(* Logix 5000 project; controller ACMI_PLC vendor 1 type 14 code 101 rev 19.11; software revision 19.01; part 17 of 18 *)
(* tags used below, declared in another part *)
   A : DINT;
   ACMI_BR_CNT : DINT;
   ACMI_Stat_Size : INT;
   ACMI_TO_CNT : DINT;
   ADCA : DINT;
   ADCB : DINT;
   B : DINT;
   Beam_MaxQ : DINT;
   Beam_MinQ : DINT;
   Beam_Q : DINT;
   BR_Stack : DINT[7200];
   BR_Stack_MAX : DINT;
   BR_Stack_Sum : DINT;
   BR_Stack_Top : DINT;
   BSSS_CLOSED : ALIAS FOR PointIONet:7:I.Pt00Data;
   BYPASS_KEY : ALIAS FOR PointIONet:5:I.Pt07Data;
   FAULT_BEAM_BL : BOOL;
   FAULT_BEAM_HI : BOOL;
   FAULT_BEAM_LO : BOOL;
   FAULT_BR_ACC : BOOL;
   FAULT_CODE : DINT;
   FAULT_QOW1 : BOOL;
   FAULT_ST1_AB_HI : BOOL;
   FAULT_ST1_AB_LO : BOOL;
   FAULT_ST1_BA_HI : BOOL;
   FAULT_ST1_BA_LO : BOOL;
   FAULT_ST1_BLA : BOOL;
   FAULT_ST1_BLB : BOOL;
   FAULT_ST1_QAT : BOOL;
   FAULT_ST2_AB_HI : BOOL;
   FAULT_ST2_AB_LO : BOOL;
   FAULT_ST2_BA_HI : BOOL;
   FAULT_ST2_BA_LO : BOOL;
   FAULT_ST2_BLA : BOOL;
   FAULT_ST2_BLB : BOOL;
   FAULT_ST2_QAT : BOOL;
   FAULT_TO_ACC : BOOL;
   FAULT_TWB : BOOL;
   FAULT_WDT : BOOL;
   Initialize : BOOL;
   LBSS_CLOSED : ALIAS FOR PointIONet:7:I.Pt01Data;
   ST1_MaxQ : DINT;
   ST1_MinQ : DINT;
   ST1_QAB : DINT;
   ST1_QBA : DINT;
   ST2_MaxQ : DINT;
   ST2_MinQ : DINT;
   ST2_QAB : DINT;
   ST2_QBA : DINT;
   ST_HI_FAULT : BOOL;
   ST_LO_FAULT : BOOL;
   ST_Size : BOOL;
   ST_Type : BOOL;
   Stack_Size : DINT;
   TO_Cntr : COUNTER;
   TO_DISABLED : ALIAS FOR PointIONet:7:I.Pt03Data;
   TO_Stack : DINT[120];
   TO_Stack_MAX : DINT;
   TO_Stack_Size : DINT;
   TO_Stack_Sum : DINT;
   TO_Stack_Top : DINT;
   TO_Status_Error : BOOL;
   Update_ST1_QAB : BOOL;
   Update_ST1_QBA : BOOL;
   Update_ST2_QAB : BOOL;
   Update_ST2_QBA : BOOL;
   Zero : DINT[7200];

        [22].Hist[3812] := 1, [22].Hist[3815] := 1, [22].Hist[3816] := 1, [22].Hist[3817] := 1, [22].Hist[3819] := 1, [22].Hist[3820] := 1, [22].Hist[3824] := 1, [22].Hist[3825] := 1, [22].Hist[3828] := 1, [22].Hist[3832] := 1, [22].Hist[3835] := 1, [22].Hist[3836] := 1, [22].Hist[3839] := 1, [22].Hist[3840] := 1, [22].Hist[3844] := 1, [22].Hist[3848] := 1, [22].Hist[3852] := 1, [22].Hist[3853] := 1, [22].Hist[3855] := 1, [22].Hist[3856] := 1, [22].Hist[3859] := 1, [22].Hist[3860] := 1, [22].Hist[3864] := 1, [22].Hist[3868] := 1, [22].Hist[3869] := 1, [22].Hist[3872] := 1, [22].Hist[3875] := 1, [22].Hist[3876] := 1, [22].Hist[3880] := 1, [22].Hist[3881] := 1, [22].Hist[3883] := 1, [22].Hist[3884] := 1, [22].Hist[3885] := 1, [22].Hist[3888] := 1, [22].Hist[3891] := 1, [22].Hist[3892] := 1, [22].Hist[3896] := 1, [22].Hist[3900] := 1, [22].Hist[3901] := 1, [22].Hist[3903] := 1, [22].Hist[3904] := 1, [22].Hist[3908] := 1, [22].Hist[3912] := 1, [22].Hist[3916] := 1, [22].Hist[3917] := 1, [22].Hist[3920] := 1, [22].Hist[3921] := 1, [22].Hist[3924] := 1, [22].Hist[3927] := 1, [22].Hist[3928] := 1, [22].Hist[3929] := 1, [22].Hist[3932] := 1, [22].Hist[3935] := 1, [22].Hist[3936] := 1, [22].Hist[3940] := 1, [22].Hist[3944] := 1, [22].Hist[3948] := 1, [22].Hist[3952] := 1, [22].Hist[3953] := 1, [22].Hist[3955] := 1,
        [22].Hist[3956] := 1, [22].Hist[3960] := 1, [22].Hist[3964] := 1, [22].Hist[3967] := 1, [22].Hist[3968] := 1, [22].Hist[3969] := 1, [22].Hist[3972] := 1, [22].Hist[3976] := 1, [22].Hist[3977] := 1, [22].Hist[3980] := 1, [22].Hist[3984] := 1, [22].Hist[3988] := 1, [22].Hist[3992] := 1, [22].Hist[3995] := 1, [22].Hist[3996] := 1, [22].Hist[4000] := 1, [22].Hist[4004] := 1, [22].Hist[4008] := 1, [22].Hist[4012] := 1, [22].Hist[4013] := 1, [22].Hist[4016] := 1, [22].Hist[4020] := 1, [22].Hist[4024] := 1, [22].Hist[4025] := 1, [22].Hist[4028] := 1, [22].Hist[4029] := 1, [22].Hist[4032] := 1, [22].Hist[4036] := 1, [22].Hist[4040] := 1, [22].Hist[4044] := 1, [22].Hist[4047] := 1, [22].Hist[4048] := 1, [22].Hist[4052] := 1, [22].Hist[4056] := 1, [22].Hist[4057] := 1, [22].Hist[4060] := 1, [22].Hist[4061] := 1, [22].Hist[4063] := 1, [22].Hist[4064] := 1, [22].Hist[4068] := 1, [22].Hist[4072] := 1, [22].Hist[4076] := 1, [22].Hist[4080] := 1, [22].Hist[4081] := 1, [22].Hist[4084] := 1, [22].Hist[4087] := 1, [22].Hist[4088] := 1, [22].Hist[4092] := 1, [22].Top := 3827, [22].Sum := 1635, [23].Hist[3] := 1, [23].Hist[5] := 1, [23].Hist[9] := 1, [23].Hist[17] := 1, [23].Hist[19] := 1, [23].Hist[29] := 1, [23].Hist[31] := 1, [23].Hist[37] := 1, [23].Hist[39] := 1, [23].Hist[41] := 1,
        [23].Hist[51] := 1, [23].Hist[55] := 1, [23].Hist[63] := 1, [23].Hist[67] := 1, [23].Hist[73] := 1, [23].Hist[77] := 1, [23].Hist[81] := 1, [23].Hist[89] := 1, [23].Hist[95] := 1, [23].Hist[107] := 1, [23].Hist[115] := 1, [23].Hist[117] := 1, [23].Hist[125] := 1, [23].Hist[127] := 1, [23].Hist[135] := 1, [23].Hist[153] := 1, [23].Hist[155] := 1, [23].Hist[165] := 1, [23].Hist[179] := 1, [23].Hist[187] := 1, [23].Hist[199] := 1, [23].Hist[213] := 1, [23].Hist[223] := 1, [23].Hist[239] := 1, [23].Hist[243] := 1, [23].Hist[251] := 1, [23].Hist[253] := 1, [23].Hist[255] := 1, [23].Hist[257] := 1, [23].Hist[261] := 1, [23].Hist[271] := 1, [23].Hist[277] := 1, [23].Hist[291] := 1, [23].Hist[293] := 1, [23].Hist[301] := 1, [23].Hist[307] := 1, [23].Hist[313] := 1, [23].Hist[317] := 1, [23].Hist[321] := 1, [23].Hist[323] := 1, [23].Hist[331] := 1, [23].Hist[337] := 1, [23].Hist[341] := 1, [23].Hist[347] := 1, [23].Hist[351] := 1, [23].Hist[353] := 1, [23].Hist[359] := 1, [23].Hist[361] := 1, [23].Hist[365] := 1, [23].Hist[367] := 1, [23].Hist[369] := 1, [23].Hist[373] := 1, [23].Hist[405] := 1, [23].Hist[413] := 1, [23].Hist[417] := 1, [23].Hist[423] := 1, [23].Hist[425] := 1, [23].Hist[429] := 1, [23].Hist[433] := 1, [23].Hist[441] := 1,
        [23].Hist[443] := 1, [23].Hist[445] := 1, [23].Hist[447] := 1, [23].Hist[459] := 1, [23].Hist[471] := 1, [23].Hist[473] := 1, [23].Hist[491] := 1, [23].Hist[501] := 1, [23].Hist[509] := 1, [23].Hist[515] := 1, [23].Hist[519] := 1, [23].Hist[527] := 1, [23].Hist[529] := 1, [23].Hist[537] := 1, [23].Hist[543] := 1, [23].Hist[547] := 1, [23].Hist[553] := 1, [23].Hist[557] := 1, [23].Hist[559] := 1, [23].Hist[567] := 1, [23].Hist[569] := 1, [23].Hist[581] := 1, [23].Hist[601] := 1, [23].Hist[611] := 1, [23].Hist[613] := 1, [23].Hist[619] := 1, [23].Hist[621] := 1, [23].Hist[629] := 1, [23].Hist[637] := 1, [23].Hist[647] := 1, [23].Hist[663] := 1, [23].Hist[669] := 1, [23].Hist[677] := 1, [23].Hist[679] := 1, [23].Hist[689] := 1, [23].Hist[691] := 1, [23].Hist[693] := 1, [23].Hist[695] := 1, [23].Hist[709] := 1, [23].Hist[723] := 1, [23].Hist[737] := 1, [23].Hist[741] := 1, [23].Hist[747] := 1, [23].Hist[749] := 1, [23].Hist[751] := 1, [23].Hist[761] := 1, [23].Hist[767] := 1, [23].Hist[773] := 1, [23].Hist[777] := 1, [23].Hist[799] := 1, [23].Hist[801] := 1, [23].Hist[825] := 1, [23].Hist[827] := 1, [23].Hist[829] := 1, [23].Hist[841] := 1, [23].Hist[847] := 1, [23].Hist[853] := 1, [23].Hist[859] := 1, [23].Hist[863] := 1, [23].Hist[865] := 1,
        [23].Hist[867] := 1, [23].Hist[875] := 1, [23].Hist[877] := 1, [23].Hist[879] := 1, [23].Hist[881] := 1, [23].Hist[883] := 1, [23].Hist[891] := 1, [23].Hist[893] := 1, [23].Hist[911] := 1, [23].Hist[923] := 1, [23].Hist[927] := 1, [23].Hist[935] := 1, [23].Hist[943] := 1, [23].Hist[945] := 1, [23].Hist[947] := 1, [23].Hist[961] := 1, [23].Hist[969] := 1, [23].Hist[973] := 1, [23].Hist[983] := 1, [23].Hist[985] := 1, [23].Hist[987] := 1, [23].Hist[995] := 1, [23].Hist[1015] := 1, [23].Hist[1021] := 1, [23].Hist[1041] := 1, [23].Hist[1045] := 1, [23].Hist[1047] := 1, [23].Hist[1049] := 1, [23].Hist[1053] := 1, [23].Hist[1057] := 1, [23].Hist[1059] := 1, [23].Hist[1061] := 1, [23].Hist[1065] := 1, [23].Hist[1073] := 1, [23].Hist[1077] := 1, [23].Hist[1079] := 1, [23].Hist[1085] := 1, [23].Hist[1093] := 1, [23].Hist[1095] := 1, [23].Hist[1101] := 1, [23].Hist[1109] := 1, [23].Hist[1125] := 1, [23].Hist[1129] := 1, [23].Hist[1135] := 1, [23].Hist[1137] := 1, [23].Hist[1141] := 1, [23].Hist[1145] := 1, [23].Hist[1149] := 1, [23].Hist[1155] := 1, [23].Hist[1167] := 1, [23].Hist[1175] := 1, [23].Hist[1181] := 1, [23].Hist[1185] := 1, [23].Hist[1195] := 1, [23].Hist[1209] := 1, [23].Hist[1217] := 1, [23].Hist[1235] := 1, [23].Hist[1237] := 1, [23].Hist[1239] := 1, [23].Hist[1245] := 1,
        [23].Hist[1257] := 1, [23].Hist[1265] := 1, [23].Hist[1269] := 1, [23].Hist[1271] := 1, [23].Hist[1277] := 1, [23].Hist[1279] := 1, [23].Hist[1281] := 1, [23].Hist[1291] := 1, [23].Hist[1299] := 1, [23].Hist[1307] := 1, [23].Hist[1325] := 1, [23].Hist[1329] := 1, [23].Hist[1335] := 1, [23].Hist[1347] := 1, [23].Hist[1349] := 1, [23].Hist[1351] := 1, [23].Hist[1357] := 1, [23].Hist[1361] := 1, [23].Hist[1365] := 1, [23].Hist[1383] := 1, [23].Hist[1389] := 1, [23].Hist[1397] := 1, [23].Hist[1401] := 1, [23].Hist[1407] := 1, [23].Hist[1411] := 1, [23].Hist[1413] := 1, [23].Hist[1419] := 1, [23].Hist[1429] := 1, [23].Hist[1437] := 1, [23].Hist[1451] := 1, [23].Hist[1469] := 1, [23].Hist[1471] := 1, [23].Hist[1477] := 1, [23].Hist[1483] := 1, [23].Hist[1487] := 1, [23].Hist[1489] := 1, [23].Hist[1491] := 1, [23].Hist[1495] := 1, [23].Hist[1497] := 1, [23].Hist[1501] := 1, [23].Hist[1511] := 1, [23].Hist[1515] := 1, [23].Hist[1517] := 1, [23].Hist[1519] := 1, [23].Hist[1521] := 1, [23].Hist[1535] := 1, [23].Hist[1539] := 1, [23].Hist[1545] := 1, [23].Hist[1547] := 1, [23].Hist[1551] := 1, [23].Hist[1555] := 1, [23].Hist[1557] := 1, [23].Hist[1559] := 1, [23].Hist[1563] := 1, [23].Hist[1565] := 1, [23].Hist[1569] := 1, [23].Hist[1581] := 1, [23].Hist[1593] := 1, [23].Hist[1605] := 1, [23].Hist[1611] := 1,
        [23].Hist[1617] := 1, [23].Hist[1627] := 1, [23].Hist[1651] := 1, [23].Hist[1653] := 1, [23].Hist[1655] := 1, [23].Hist[1669] := 1, [23].Hist[1677] := 1, [23].Hist[1679] := 1, [23].Hist[1681] := 1, [23].Hist[1683] := 1, [23].Hist[1685] := 1, [23].Hist[1691] := 1, [23].Hist[1697] := 1, [23].Hist[1709] := 1, [23].Hist[1715] := 1, [23].Hist[1717] := 1, [23].Hist[1721] := 1, [23].Hist[1731] := 1, [23].Hist[1737] := 1, [23].Hist[1741] := 1, [23].Hist[1747] := 1, [23].Hist[1753] := 1, [23].Hist[1769] := 1, [23].Hist[1771] := 1, [23].Hist[1779] := 1, [23].Hist[1783] := 1, [23].Hist[1785] := 1, [23].Hist[1793] := 1, [23].Hist[1805] := 1, [23].Hist[1807] := 1, [23].Hist[1811] := 1, [23].Hist[1819] := 1, [23].Hist[1821] := 1, [23].Hist[1825] := 1, [23].Hist[1827] := 1, [23].Hist[1833] := 1, [23].Hist[1839] := 1, [23].Hist[1843] := 1, [23].Hist[1849] := 1, [23].Hist[1851] := 1, [23].Hist[1857] := 1, [23].Hist[1863] := 1, [23].Hist[1877] := 1, [23].Hist[1879] := 1, [23].Hist[1881] := 1, [23].Hist[1883] := 1, [23].Hist[1885] := 1, [23].Hist[1891] := 1, [23].Hist[1893] := 1, [23].Hist[1901] := 1, [23].Hist[1903] := 1, [23].Hist[1905] := 1, [23].Hist[1921] := 1, [23].Hist[1931] := 1, [23].Hist[1933] := 1, [23].Hist[1935] := 1, [23].Hist[1945] := 1, [23].Hist[1949] := 1, [23].Hist[1953] := 1, [23].Hist[1959] := 1,
        [23].Hist[1975] := 1, [23].Hist[1977] := 1, [23].Hist[1999] := 1, [23].Hist[2005] := 1, [23].Hist[2017] := 1, [23].Hist[2019] := 1, [23].Hist[2043] := 1, [23].Hist[2061] := 1, [23].Hist[2065] := 1, [23].Hist[2071] := 1, [23].Hist[2075] := 1, [23].Hist[2079] := 1, [23].Hist[2085] := 1, [23].Hist[2089] := 1, [23].Hist[2107] := 1, [23].Hist[2111] := 1, [23].Hist[2119] := 1, [23].Hist[2125] := 1, [23].Hist[2127] := 1, [23].Hist[2129] := 1, [23].Hist[2131] := 1, [23].Hist[2139] := 1, [23].Hist[2151] := 1, [23].Hist[2157] := 1, [23].Hist[2173] := 1, [23].Hist[2175] := 1, [23].Hist[2183] := 1, [23].Hist[2185] := 1, [23].Hist[2195] := 1, [23].Hist[2197] := 1, [23].Hist[2223] := 1, [23].Hist[2229] := 1, [23].Hist[2231] := 1, [23].Hist[2233] := 1, [23].Hist[2241] := 1, [23].Hist[2243] := 1, [23].Hist[2245] := 1, [23].Hist[2249] := 1, [23].Hist[2251] := 1, [23].Hist[2253] := 1, [23].Hist[2255] := 1, [23].Hist[2257] := 1, [23].Hist[2259] := 1, [23].Hist[2263] := 1, [23].Hist[2271] := 1, [23].Hist[2273] := 1, [23].Hist[2289] := 1, [23].Hist[2311] := 1, [23].Hist[2313] := 1, [23].Hist[2325] := 1, [23].Hist[2327] := 1, [23].Hist[2339] := 1, [23].Hist[2355] := 1, [23].Hist[2357] := 1, [23].Hist[2365] := 1, [23].Hist[2367] := 1, [23].Hist[2371] := 1, [23].Hist[2379] := 1, [23].Hist[2387] := 1, [23].Hist[2397] := 1,
        [23].Hist[2409] := 1, [23].Hist[2413] := 1, [23].Hist[2421] := 1, [23].Hist[2425] := 1, [23].Hist[2427] := 1, [23].Hist[2429] := 1, [23].Hist[2431] := 1, [23].Hist[2437] := 1, [23].Hist[2441] := 1, [23].Hist[2445] := 1, [23].Hist[2459] := 1, [23].Hist[2461] := 1, [23].Hist[2477] := 1, [23].Hist[2483] := 1, [23].Hist[2487] := 1, [23].Hist[2497] := 1, [23].Hist[2509] := 1, [23].Hist[2513] := 1, [23].Hist[2519] := 1, [23].Hist[2523] := 1, [23].Hist[2531] := 1, [23].Hist[2533] := 1, [23].Hist[2537] := 1, [23].Hist[2539] := 1, [23].Hist[2549] := 1, [23].Hist[2555] := 1, [23].Hist[2589] := 1, [23].Hist[2597] := 1, [23].Hist[2601] := 1, [23].Hist[2609] := 1, [23].Hist[2615] := 1, [23].Hist[2625] := 1, [23].Hist[2631] := 1, [23].Hist[2635] := 1, [23].Hist[2637] := 1, [23].Hist[2643] := 1, [23].Hist[2647] := 1, [23].Hist[2657] := 1, [23].Hist[2671] := 1, [23].Hist[2679] := 1, [23].Hist[2683] := 1, [23].Hist[2685] := 1, [23].Hist[2689] := 1, [23].Hist[2691] := 1, [23].Hist[2693] := 1, [23].Hist[2695] := 1, [23].Hist[2719] := 1, [23].Hist[2721] := 1, [23].Hist[2723] := 1, [23].Hist[2739] := 1, [23].Hist[2741] := 1, [23].Hist[2757] := 1, [23].Hist[2761] := 1, [23].Hist[2765] := 1, [23].Hist[2767] := 1, [23].Hist[2781] := 1, [23].Hist[2785] := 1, [23].Hist[2787] := 1, [23].Hist[2801] := 1, [23].Hist[2809] := 1,
        [23].Hist[2811] := 1, [23].Hist[2819] := 1, [23].Hist[2821] := 1, [23].Hist[2837] := 1, [23].Hist[2841] := 1, [23].Hist[2843] := 1, [23].Hist[2861] := 1, [23].Hist[2863] := 1, [23].Hist[2865] := 1, [23].Hist[2875] := 1, [23].Hist[2877] := 1, [23].Hist[2883] := 1, [23].Hist[2887] := 1, [23].Hist[2889] := 1, [23].Hist[2899] := 1, [23].Hist[2901] := 1, [23].Hist[2903] := 1, [23].Hist[2909] := 1, [23].Hist[2921] := 1, [23].Hist[2925] := 1, [23].Hist[2929] := 1, [23].Hist[2937] := 1, [23].Hist[2939] := 1, [23].Hist[2951] := 1, [23].Hist[2955] := 1, [23].Hist[2963] := 1, [23].Hist[2975] := 1, [23].Hist[2981] := 1, [23].Hist[2989] := 1, [23].Hist[2993] := 1, [23].Hist[2995] := 1, [23].Hist[2999] := 1, [23].Hist[3009] := 1, [23].Hist[3019] := 1, [23].Hist[3025] := 1, [23].Hist[3037] := 1, [23].Hist[3053] := 1, [23].Hist[3059] := 1, [23].Hist[3069] := 1, [23].Hist[3079] := 1, [23].Hist[3095] := 1, [23].Hist[3101] := 1, [23].Hist[3105] := 1, [23].Hist[3107] := 1, [23].Hist[3109] := 1, [23].Hist[3111] := 1, [23].Hist[3113] := 1, [23].Hist[3133] := 1, [23].Hist[3141] := 1, [23].Hist[3145] := 1, [23].Hist[3153] := 1, [23].Hist[3157] := 1, [23].Hist[3165] := 1, [23].Hist[3167] := 1, [23].Hist[3177] := 1, [23].Hist[3183] := 1, [23].Hist[3189] := 1, [23].Hist[3199] := 1, [23].Hist[3201] := 1, [23].Hist[3205] := 1,
        [23].Hist[3211] := 1, [23].Hist[3213] := 1, [23].Hist[3221] := 1, [23].Hist[3231] := 1, [23].Hist[3233] := 1, [23].Hist[3235] := 1, [23].Hist[3245] := 1, [23].Hist[3259] := 1, [23].Hist[3265] := 1, [23].Hist[3275] := 1, [23].Hist[3281] := 1, [23].Hist[3283] := 1, [23].Hist[3287] := 1, [23].Hist[3289] := 1, [23].Hist[3293] := 1, [23].Hist[3295] := 1, [23].Hist[3303] := 1, [23].Hist[3305] := 1, [23].Hist[3309] := 1, [23].Hist[3311] := 1, [23].Hist[3315] := 1, [23].Hist[3319] := 1, [23].Hist[3327] := 1, [23].Hist[3335] := 1, [23].Hist[3343] := 1, [23].Hist[3351] := 1, [23].Hist[3353] := 1, [23].Hist[3361] := 1, [23].Hist[3363] := 1, [23].Hist[3365] := 1, [23].Hist[3367] := 1, [23].Hist[3369] := 1, [23].Hist[3373] := 1, [23].Hist[3379] := 1, [23].Hist[3387] := 1, [23].Hist[3401] := 1, [23].Hist[3409] := 1, [23].Hist[3421] := 1, [23].Hist[3441] := 1, [23].Hist[3447] := 1, [23].Hist[3453] := 1, [23].Hist[3475] := 1, [23].Hist[3479] := 1, [23].Hist[3485] := 1, [23].Hist[3505] := 1, [23].Hist[3507] := 1, [23].Hist[3527] := 1, [23].Hist[3529] := 1, [23].Hist[3535] := 1, [23].Hist[3545] := 1, [23].Hist[3571] := 1, [23].Hist[3577] := 1, [23].Hist[3585] := 1, [23].Hist[3591] := 1, [23].Hist[3593] := 1, [23].Hist[3601] := 1, [23].Hist[3611] := 1, [23].Hist[3613] := 1, [23].Hist[3625] := 1, [23].Hist[3639] := 1,
        [23].Hist[3659] := 1, [23].Hist[3663] := 1, [23].Hist[3671] := 1, [23].Hist[3673] := 1, [23].Hist[3679] := 1, [23].Hist[3687] := 1, [23].Hist[3689] := 1, [23].Hist[3707] := 1, [23].Hist[3713] := 1, [23].Hist[3727] := 1, [23].Hist[3737] := 1, [23].Hist[3739] := 1, [23].Hist[3747] := 1, [23].Hist[3749] := 1, [23].Hist[3753] := 1, [23].Hist[3757] := 1, [23].Hist[3761] := 1, [23].Hist[3763] := 1, [23].Hist[3771] := 1, [23].Hist[3787] := 1, [23].Hist[3789] := 1, [23].Hist[3791] := 1, [23].Hist[3795] := 1, [23].Hist[3811] := 1, [23].Hist[3815] := 1, [23].Hist[3817] := 1, [23].Hist[3819] := 1, [23].Hist[3825] := 1, [23].Hist[3835] := 1, [23].Hist[3839] := 1, [23].Hist[3853] := 1, [23].Hist[3855] := 1, [23].Hist[3859] := 1, [23].Hist[3869] := 1, [23].Hist[3875] := 1, [23].Hist[3881] := 1, [23].Hist[3883] := 1, [23].Hist[3885] := 1, [23].Hist[3891] := 1, [23].Hist[3901] := 1, [23].Hist[3903] := 1, [23].Hist[3917] := 1, [23].Hist[3921] := 1, [23].Hist[3927] := 1, [23].Hist[3929] := 1, [23].Hist[3935] := 1, [23].Hist[3953] := 1, [23].Hist[3955] := 1, [23].Hist[3967] := 1, [23].Hist[3969] := 1, [23].Hist[3977] := 1, [23].Hist[3995] := 1, [23].Hist[4013] := 1, [23].Hist[4025] := 1, [23].Hist[4029] := 1, [23].Hist[4047] := 1, [23].Hist[4057] := 1, [23].Hist[4061] := 1, [23].Hist[4063] := 1, [23].Hist[4081] := 1,
        [23].Hist[4087] := 1, [23].Top := 3827, [23].Sum := 611);
   Bx : DINT := 58; {access Read Only}
   Data_Type : BOOL := 1;
   DrdyTimer : TIMER := (PRE := 500, EN := 1, TT := 1);
   DrdyWDT : DINT := 220;
   ev_num : COUNTER := (ACC := 945682714, DN := 1);
   Fit_Linear_1 : DINT := 91341; {constant}
   Fit_Linear_2 : DINT := 10000; {constant}
   Fit_Off : DINT := 21; {constant}
   Fit_Quad_1 : DINT := 273; {constant}
   Fit_Quad_2 : DINT := 1000000; {constant}
   Hist : BOOL[4096] := ([956] := 1, [1408] := 1, [2824] := 1, [3245] := 1, [3333] := 1, [3825] := 1, [4017] := 1);
   index : DINT;
   NewData : BOOL;
   Q : DINT := 19062;
   QIW : BOOL := 1;
   Qlinear : DINT := 18189;
   QOW_FailSafe : TIMER := (PRE := 2000, ACC := 380); {access Read Only}
   QOW_Latch : BOOL := 1;
   Qquad : DINT := 866;
   ReadData : BOOL;
   Relay_Status : ALIAS FOR PointIONet:5:I.Pt04Data;
   Safety_Shutters : BOOL;
   ST1AB_ADCA : DINT := 2047; {access Read Only}
   ST1AB_ADCB : DINT := 62; {access Read Only}
   ST1BA_ADCA : DINT := 49; {access Read Only}
   ST1BA_ADCB : DINT := 2047; {access Read Only}
   ST2AB_ADCA : DINT := 2047; {access Read Only}
   ST2AB_ADCB : DINT := 58; {access Read Only}
   ST2BA_ADCA : DINT := 51; {access Read Only}
   ST2BA_ADCB : DINT := 2047; {access Read Only}
   Stack_Data : DINT := 180;
   STQ : DINT := 19062; {access Read Only}
   STQmax : DINT := 16400; {access Read Only}
   STQmin : DINT := 15400; {access Read Only}
   Sum : INT := 7;
   Toggle : BitStat[12];
   Top : INT := 361;
   TWB_FailSafe : TIMER := (PRE := 2000, ACC := 20); {access Read Only}
   TWB_Latch : BOOL;
   Update_Latch : BOOL := 1; {access Read Only}
   Update_Unlatch : BOOL; {access Read Only}
   w1 : DINT; {access Read Only}
   w2 : DINT; {access Read Only}
   WDT_Event_Limit : DINT := 265; {constant, access Read Only}
   x : DINT := 2047;
   y : DINT := 58;
   z : DINT := 1989;
   z2 : DINT;
END_VAR

ROUTINE Bit_Toggle   (* ladder *)
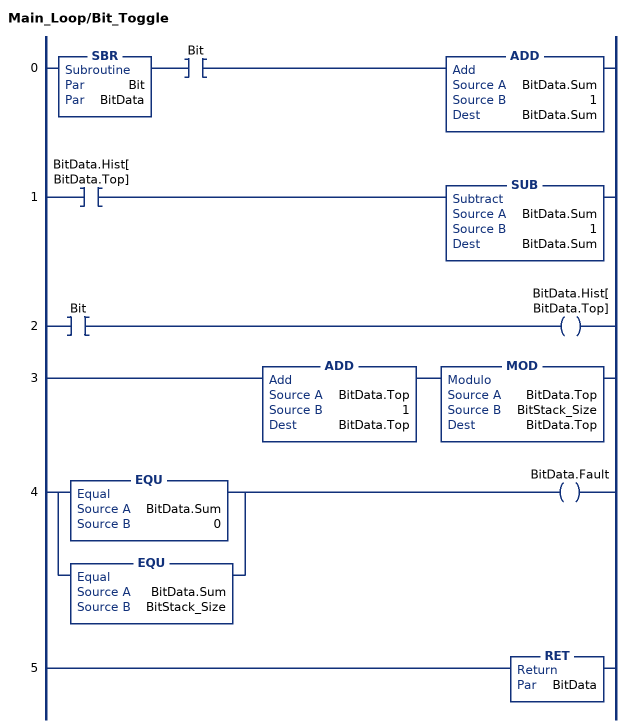
   [picture p14: Main_Loop/Bit_Toggle rungs 0-5]
   0: SBR(Bit,BitData)XIC(Bit)ADD(BitData.Sum,1,BitData.Sum);
   1: XIC(BitData.Hist[BitData.Top])SUB(BitData.Sum,1,BitData.Sum);
   2: XIC(Bit)OTE(BitData.Hist[BitData.Top]);
   3: ADD(BitData.Top,1,BitData.Top)MOD(BitData.Top,BitStack_Size,BitData.Top);
   4: [EQU(BitData.Sum,0) ,EQU(BitData.Sum,BitStack_Size) ]OTE(BitData.Fault);
   5: RET(BitData);
END_ROUTINE

ROUTINE Calc_Q   (* ladder *)
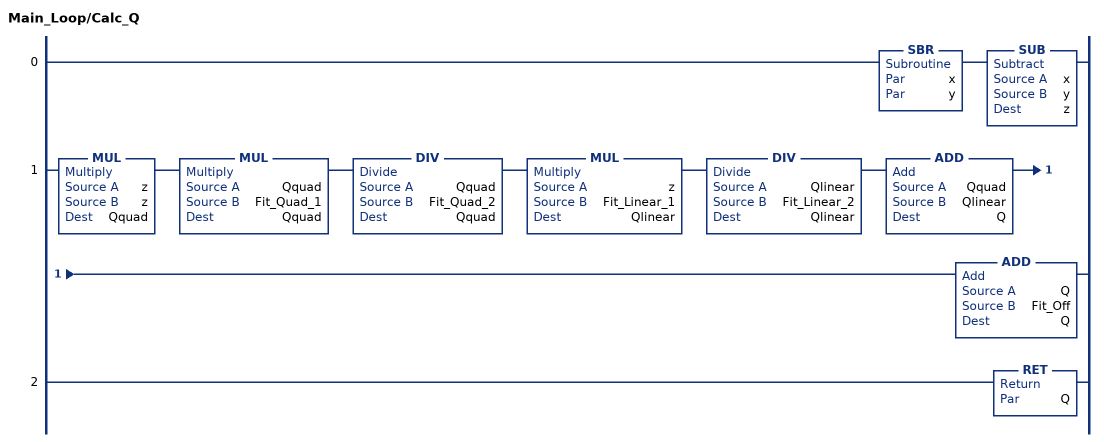
   0: SBR(x,y)SUB(x,y,z);
   1: MUL(z,z,Qquad)MUL(Qquad,Fit_Quad_1,Qquad)DIV(Qquad,Fit_Quad_2,Qquad)MUL(z,Fit_Linear_1,Qlinear)DIV(Qlinear,Fit_Linear_2,Qlinear)ADD(Qquad,Qlinear,Q)ADD(Q,Fit_Off,Q);
   2: RET(Q);
END_ROUTINE

ROUTINE MainRoutine   (* ladder *)
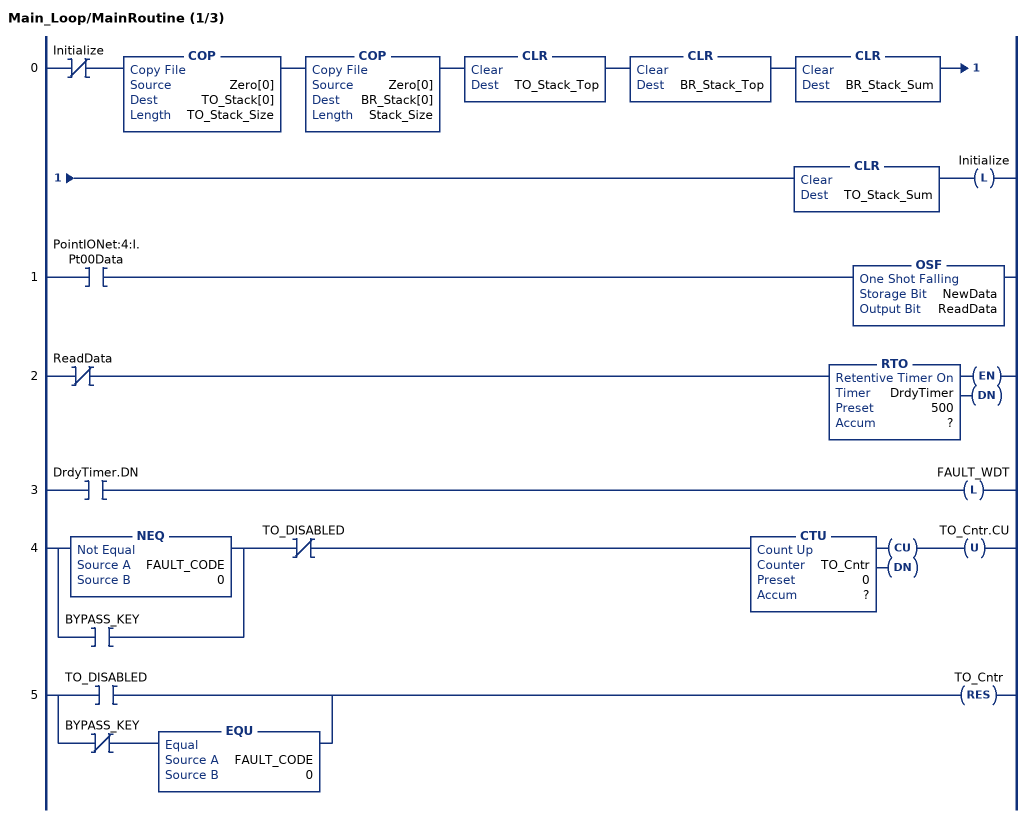
   0: XIO(Initialize)COP(Zero[0],TO_Stack[0],TO_Stack_Size)COP(Zero[0],BR_Stack[0],Stack_Size)CLR(TO_Stack_Top)CLR(BR_Stack_Top)CLR(BR_Stack_Sum)CLR(TO_Stack_Sum)OTL(Initialize);
   1: XIC(PointIONet:4:I.Pt00Data)OSF(NewData,ReadData);
   2: XIO(ReadData)RTO(DrdyTimer,?,?);
   3: XIC(DrdyTimer.DN)OTL(FAULT_WDT);
   4: [NEQ(FAULT_CODE,0) ,XIC(BYPASS_KEY) ]XIO(TO_DISABLED)CTU(TO_Cntr,?,?)OTU(TO_Cntr.CU);
   5: [XIC(TO_DISABLED) ,XIO(BYPASS_KEY) EQU(FAULT_CODE,0) ]RES(TO_Cntr);
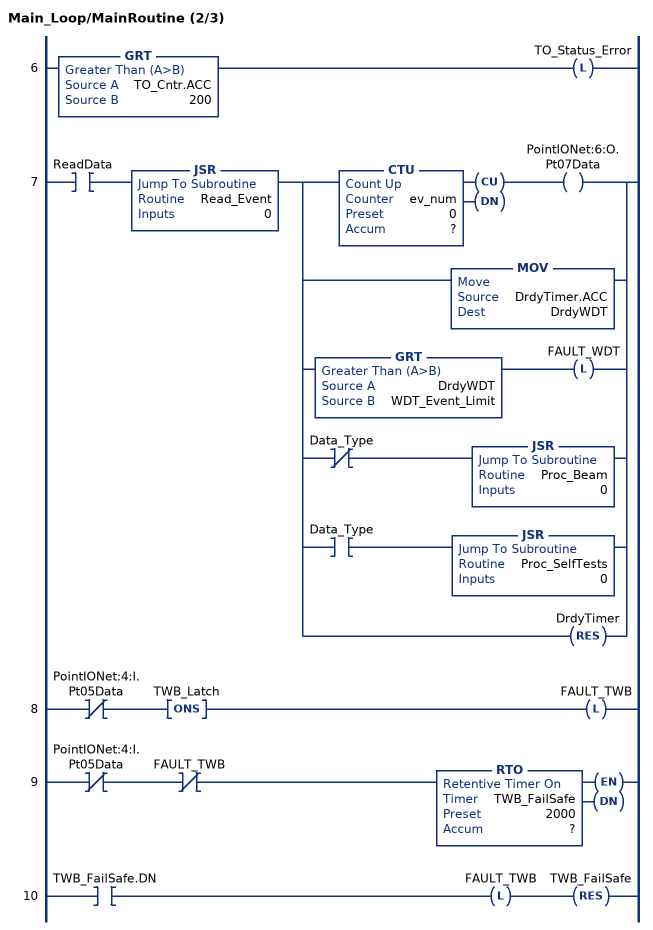
   6: GRT(TO_Cntr.ACC,200)OTL(TO_Status_Error);
   7: XIC(ReadData)JSR(Read_Event,0)[CTU(ev_num,?,?) OTE(PointIONet:6:O.Pt07Data) ,MOV(DrdyTimer.ACC,DrdyWDT) ,GRT(DrdyWDT,WDT_Event_Limit) OTL(FAULT_WDT) ,XIO(Data_Type) JSR(Proc_Beam,0) ,XIC(Data_Type) JSR(Proc_SelfTests,0) ,RES(DrdyTimer) ];
   8: XIO(PointIONet:4:I.Pt05Data)ONS(TWB_Latch)OTL(FAULT_TWB);
   9: XIO(PointIONet:4:I.Pt05Data)XIO(FAULT_TWB)RTO(TWB_FailSafe,?,?);
   10: XIC(TWB_FailSafe.DN)OTL(FAULT_TWB)RES(TWB_FailSafe);
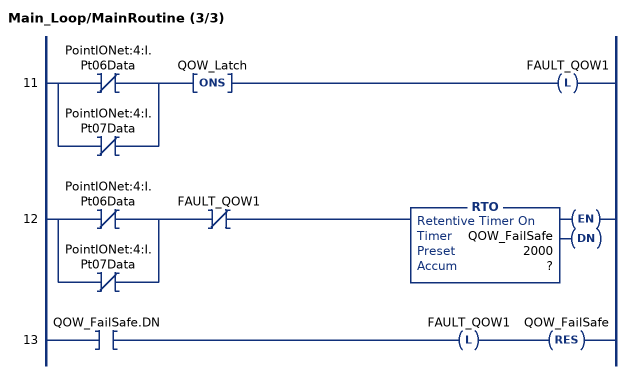
   11: [XIO(PointIONet:4:I.Pt06Data) ,XIO(PointIONet:4:I.Pt07Data) ]ONS(QOW_Latch)OTL(FAULT_QOW1);
   12: [XIO(PointIONet:4:I.Pt06Data) ,XIO(PointIONet:4:I.Pt07Data) ]XIO(FAULT_QOW1)RTO(QOW_FailSafe,?,?);
   13: XIC(QOW_FailSafe.DN)OTL(FAULT_QOW1)RES(QOW_FailSafe);
END_ROUTINE

ROUTINE Proc_Beam   (* ladder *)
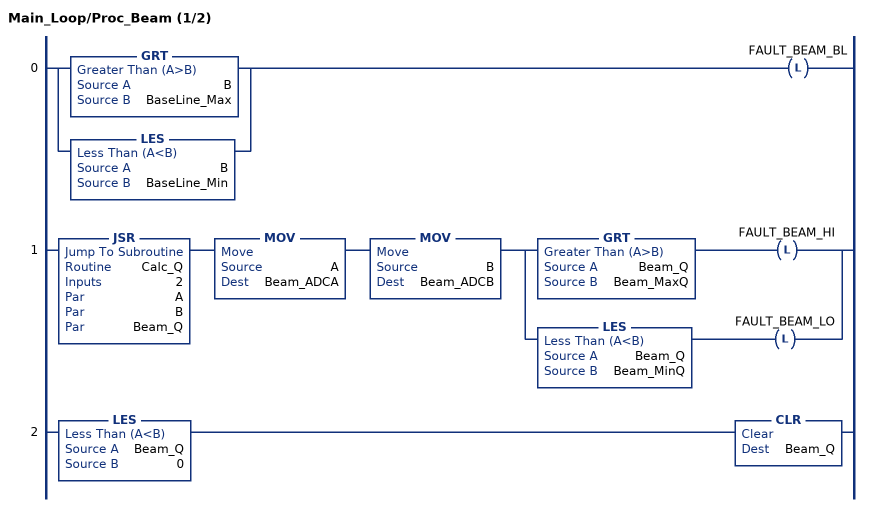
   0: [GRT(B,BaseLine_Max) ,LES(B,BaseLine_Min) ]OTL(FAULT_BEAM_BL);
   1: JSR(Calc_Q,2,A,B,Beam_Q)MOV(A,Beam_ADCA)MOV(B,Beam_ADCB)[GRT(Beam_Q,Beam_MaxQ) OTL(FAULT_BEAM_HI) ,LES(Beam_Q,Beam_MinQ) OTL(FAULT_BEAM_LO) ];
   2: LES(Beam_Q,0)CLR(Beam_Q);
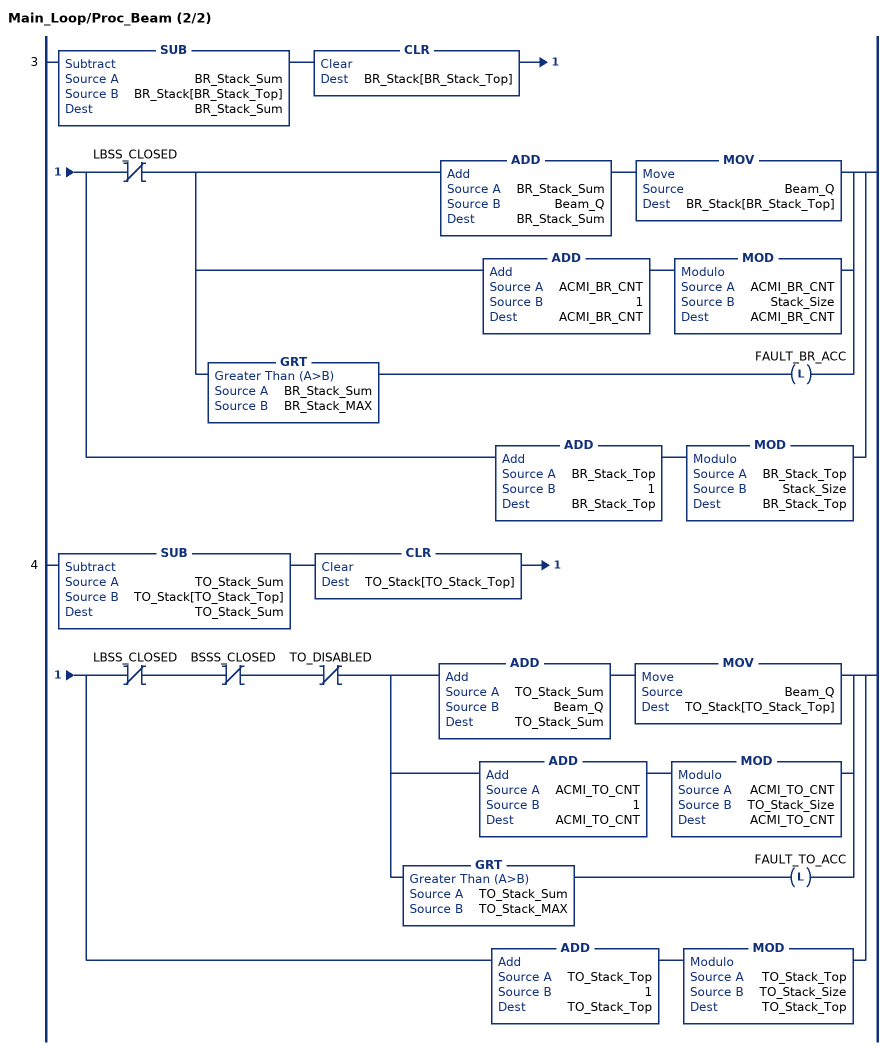
   3: SUB(BR_Stack_Sum,BR_Stack[BR_Stack_Top],BR_Stack_Sum)CLR(BR_Stack[BR_Stack_Top])[XIO(LBSS_CLOSED) [ADD(BR_Stack_Sum,Beam_Q,BR_Stack_Sum) MOV(Beam_Q,BR_Stack[BR_Stack_Top]) ,ADD(ACMI_BR_CNT,1,ACMI_BR_CNT) MOD(ACMI_BR_CNT,Stack_Size,ACMI_BR_CNT) ,GRT(BR_Stack_Sum,BR_Stack_MAX) OTL(FAULT_BR_ACC) ] ,ADD(BR_Stack_Top,1,BR_Stack_Top) MOD(BR_Stack_Top,Stack_Size,BR_Stack_Top) ];
   4: SUB(TO_Stack_Sum,TO_Stack[TO_Stack_Top],TO_Stack_Sum)CLR(TO_Stack[TO_Stack_Top])[XIO(LBSS_CLOSED) XIO(BSSS_CLOSED) XIO(TO_DISABLED) [ADD(TO_Stack_Sum,Beam_Q,TO_Stack_Sum) MOV(Beam_Q,TO_Stack[TO_Stack_Top]) ,ADD(ACMI_TO_CNT,1,ACMI_TO_CNT) MOD(ACMI_TO_CNT,TO_Stack_Size,ACMI_TO_CNT) ,GRT(TO_Stack_Sum,TO_Stack_MAX) OTL(FAULT_TO_ACC) ] ,ADD(TO_Stack_Top,1,TO_Stack_Top) MOD(TO_Stack_Top,TO_Stack_Size,TO_Stack_Top) ];
END_ROUTINE

ROUTINE Proc_SelfTests   (* ladder *)
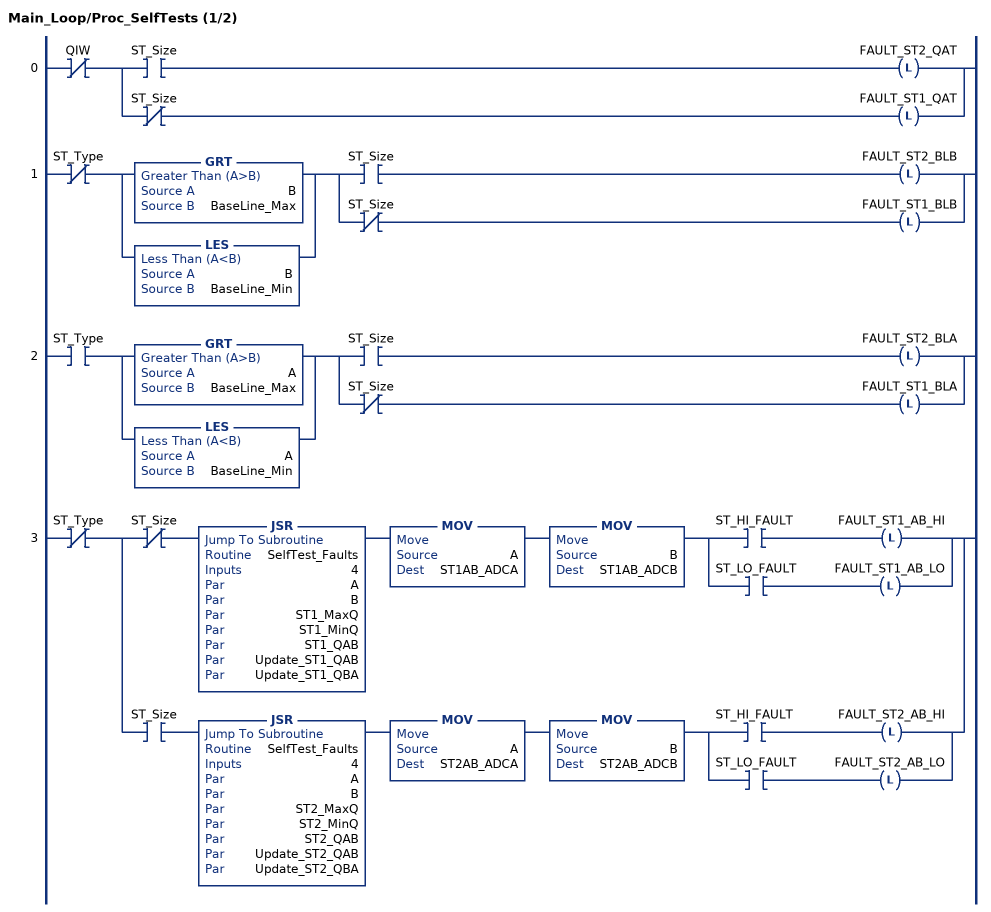
   0: XIO(QIW)[XIC(ST_Size) OTL(FAULT_ST2_QAT) ,XIO(ST_Size) OTL(FAULT_ST1_QAT) ];
   1: XIO(ST_Type)[GRT(B,BaseLine_Max) ,LES(B,BaseLine_Min) ][XIC(ST_Size) OTL(FAULT_ST2_BLB) ,XIO(ST_Size) OTL(FAULT_ST1_BLB) ];
   2: XIC(ST_Type)[GRT(A,BaseLine_Max) ,LES(A,BaseLine_Min) ][XIC(ST_Size) OTL(FAULT_ST2_BLA) ,XIO(ST_Size) OTL(FAULT_ST1_BLA) ];
   3: XIO(ST_Type)[XIO(ST_Size) JSR(SelfTest_Faults,4,A,B,ST1_MaxQ,ST1_MinQ,ST1_QAB,Update_ST1_QAB,Update_ST1_QBA) MOV(A,ST1AB_ADCA) MOV(B,ST1AB_ADCB) [XIC(ST_HI_FAULT) OTL(FAULT_ST1_AB_HI) ,XIC(ST_LO_FAULT) OTL(FAULT_ST1_AB_LO) ] ,XIC(ST_Size) JSR(SelfTest_Faults,4,A,B,ST2_MaxQ,ST2_MinQ,ST2_QAB,Update_ST2_QAB,Update_ST2_QBA) MOV(A,ST2AB_ADCA) MOV(B,ST2AB_ADCB) [XIC(ST_HI_FAULT) OTL(FAULT_ST2_AB_HI) ,XIC(ST_LO_FAULT) OTL(FAULT_ST2_AB_LO) ] ];
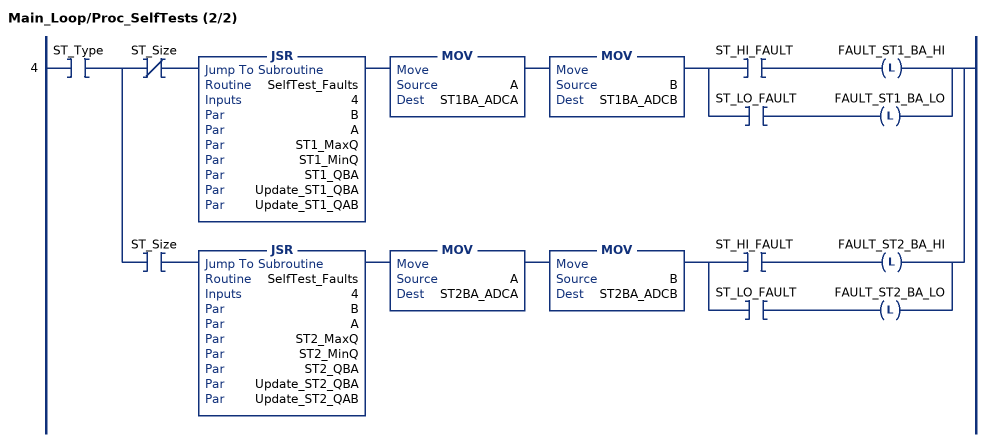
   4: XIC(ST_Type)[XIO(ST_Size) JSR(SelfTest_Faults,4,B,A,ST1_MaxQ,ST1_MinQ,ST1_QBA,Update_ST1_QBA,Update_ST1_QAB) MOV(A,ST1BA_ADCA) MOV(B,ST1BA_ADCB) [XIC(ST_HI_FAULT) OTL(FAULT_ST1_BA_HI) ,XIC(ST_LO_FAULT) OTL(FAULT_ST1_BA_LO) ] ,XIC(ST_Size) JSR(SelfTest_Faults,4,B,A,ST2_MaxQ,ST2_MinQ,ST2_QBA,Update_ST2_QBA,Update_ST2_QAB) MOV(A,ST2BA_ADCA) MOV(B,ST2BA_ADCB) [XIC(ST_HI_FAULT) OTL(FAULT_ST2_BA_HI) ,XIC(ST_LO_FAULT) OTL(FAULT_ST2_BA_LO) ] ];
END_ROUTINE

ROUTINE Read_Event   (* ladder *)
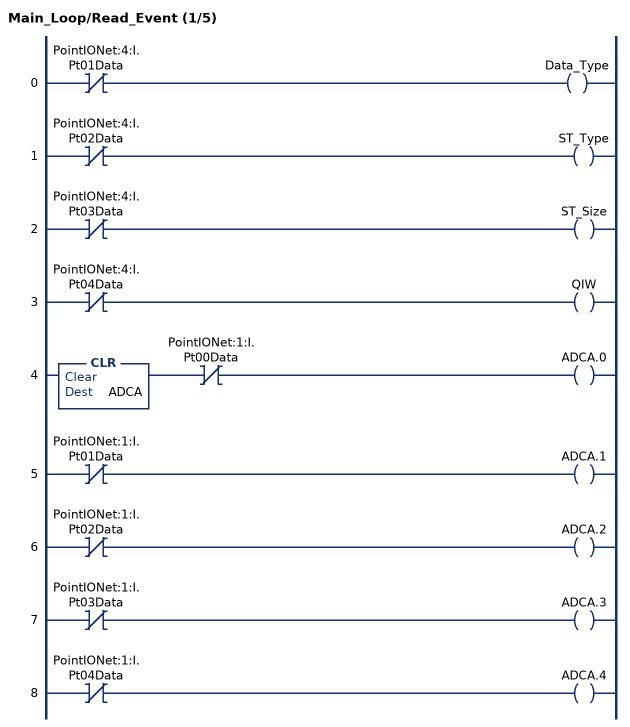
   0: XIO(PointIONet:4:I.Pt01Data)OTE(Data_Type);
   1: XIO(PointIONet:4:I.Pt02Data)OTE(ST_Type);
   2: XIO(PointIONet:4:I.Pt03Data)OTE(ST_Size);
   3: XIO(PointIONet:4:I.Pt04Data)OTE(QIW);
   4: CLR(ADCA)XIO(PointIONet:1:I.Pt00Data)OTE(ADCA.0);
   5: XIO(PointIONet:1:I.Pt01Data)OTE(ADCA.1);
   6: XIO(PointIONet:1:I.Pt02Data)OTE(ADCA.2);
   7: XIO(PointIONet:1:I.Pt03Data)OTE(ADCA.3);
   8: XIO(PointIONet:1:I.Pt04Data)OTE(ADCA.4);
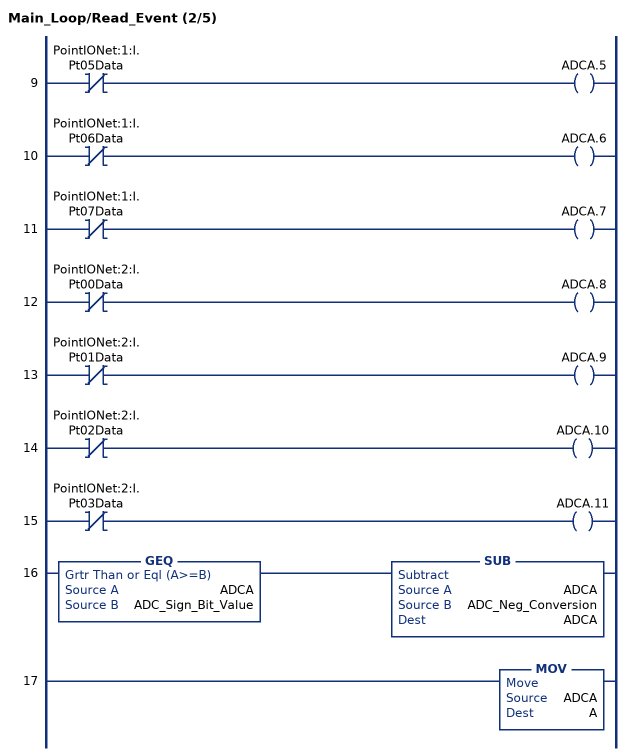
   9: XIO(PointIONet:1:I.Pt05Data)OTE(ADCA.5);
   10: XIO(PointIONet:1:I.Pt06Data)OTE(ADCA.6);
   11: XIO(PointIONet:1:I.Pt07Data)OTE(ADCA.7);
   12: XIO(PointIONet:2:I.Pt00Data)OTE(ADCA.8);
   13: XIO(PointIONet:2:I.Pt01Data)OTE(ADCA.9);
   14: XIO(PointIONet:2:I.Pt02Data)OTE(ADCA.10);
   15: XIO(PointIONet:2:I.Pt03Data)OTE(ADCA.11);
   16: GEQ(ADCA,ADC_Sign_Bit_Value)SUB(ADCA,ADC_Neg_Conversion,ADCA);
   17: MOV(ADCA,A);
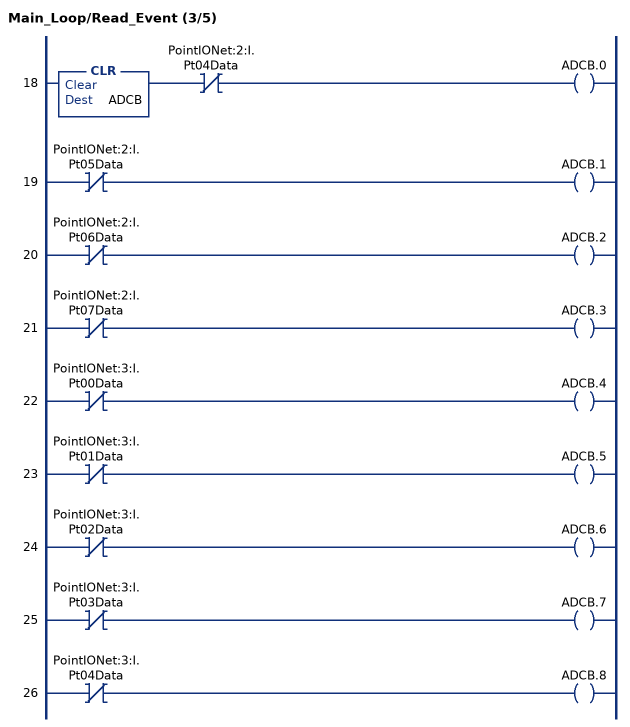
   18: CLR(ADCB)XIO(PointIONet:2:I.Pt04Data)OTE(ADCB.0);
   19: XIO(PointIONet:2:I.Pt05Data)OTE(ADCB.1);
   20: XIO(PointIONet:2:I.Pt06Data)OTE(ADCB.2);
   21: XIO(PointIONet:2:I.Pt07Data)OTE(ADCB.3);
   22: XIO(PointIONet:3:I.Pt00Data)OTE(ADCB.4);
   23: XIO(PointIONet:3:I.Pt01Data)OTE(ADCB.5);
   24: XIO(PointIONet:3:I.Pt02Data)OTE(ADCB.6);
   25: XIO(PointIONet:3:I.Pt03Data)OTE(ADCB.7);
   26: XIO(PointIONet:3:I.Pt04Data)OTE(ADCB.8);
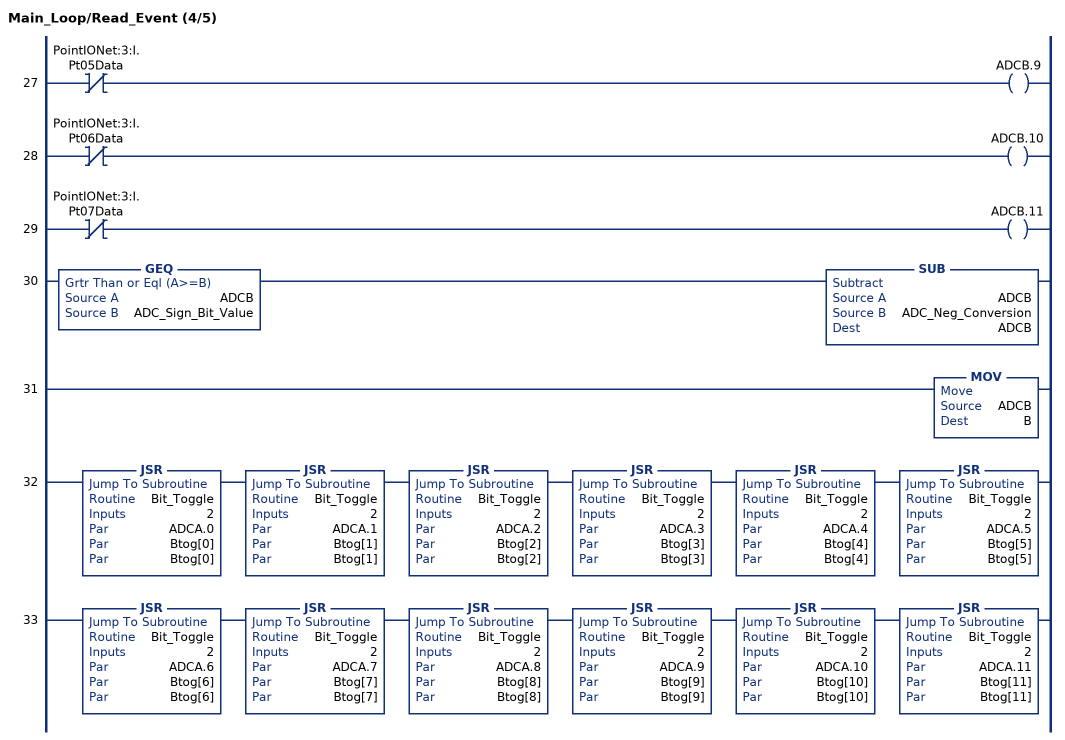
   27: XIO(PointIONet:3:I.Pt05Data)OTE(ADCB.9);
   28: XIO(PointIONet:3:I.Pt06Data)OTE(ADCB.10);
   29: XIO(PointIONet:3:I.Pt07Data)OTE(ADCB.11);
   30: GEQ(ADCB,ADC_Sign_Bit_Value)SUB(ADCB,ADC_Neg_Conversion,ADCB);
   31: MOV(ADCB,B);
   32: JSR(Bit_Toggle,2,ADCA.0,Btog[0],Btog[0])JSR(Bit_Toggle,2,ADCA.1,Btog[1],Btog[1])JSR(Bit_Toggle,2,ADCA.2,Btog[2],Btog[2])JSR(Bit_Toggle,2,ADCA.3,Btog[3],Btog[3])JSR(Bit_Toggle,2,ADCA.4,Btog[4],Btog[4])JSR(Bit_Toggle,2,ADCA.5,Btog[5],Btog[5]);
   33: JSR(Bit_Toggle,2,ADCA.6,Btog[6],Btog[6])JSR(Bit_Toggle,2,ADCA.7,Btog[7],Btog[7])JSR(Bit_Toggle,2,ADCA.8,Btog[8],Btog[8])JSR(Bit_Toggle,2,ADCA.9,Btog[9],Btog[9])JSR(Bit_Toggle,2,ADCA.10,Btog[10],Btog[10])JSR(Bit_Toggle,2,ADCA.11,Btog[11],Btog[11]);
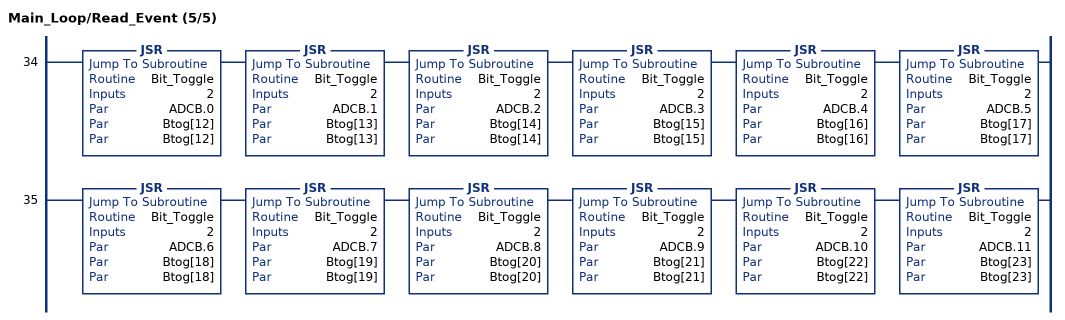
   34: JSR(Bit_Toggle,2,ADCB.0,Btog[12],Btog[12])JSR(Bit_Toggle,2,ADCB.1,Btog[13],Btog[13])JSR(Bit_Toggle,2,ADCB.2,Btog[14],Btog[14])JSR(Bit_Toggle,2,ADCB.3,Btog[15],Btog[15])JSR(Bit_Toggle,2,ADCB.4,Btog[16],Btog[16])JSR(Bit_Toggle,2,ADCB.5,Btog[17],Btog[17]);
   35: JSR(Bit_Toggle,2,ADCB.6,Btog[18],Btog[18])JSR(Bit_Toggle,2,ADCB.7,Btog[19],Btog[19])JSR(Bit_Toggle,2,ADCB.8,Btog[20],Btog[20])JSR(Bit_Toggle,2,ADCB.9,Btog[21],Btog[21])JSR(Bit_Toggle,2,ADCB.10,Btog[22],Btog[22])JSR(Bit_Toggle,2,ADCB.11,Btog[23],Btog[23]);
END_ROUTINE

ROUTINE SelfTest_Faults   (* ladder *)
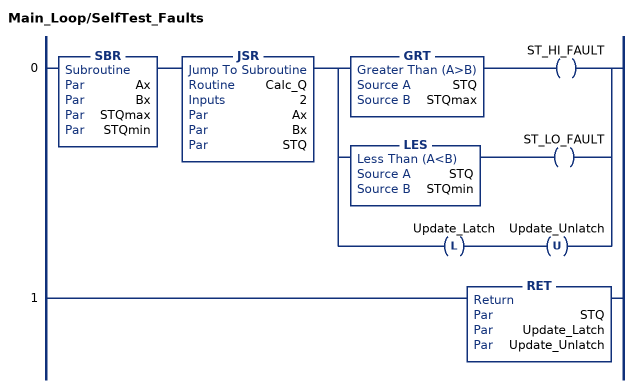
   0: SBR(Ax,Bx,STQmax,STQmin)JSR(Calc_Q,2,Ax,Bx,STQ)[GRT(STQ,STQmax) OTE(ST_HI_FAULT) ,LES(STQ,STQmin) OTE(ST_LO_FAULT) ,OTL(Update_Latch) OTU(Update_Unlatch) ];
   1: RET(STQ,Update_Latch,Update_Unlatch);
END_ROUTINE
END_PROGRAM

PROGRAM MainProgram   (* main routine Self_Test_Stats *)
VAR
   A_AVG : REAL := 2047.0;
   A_HIST : DINT[50] := ([0] := 2047, [1] := 2047, [2] := 2047, [3] := 2047, [4] := 2047, [5] := 2047, [6] := 2047, [7] := 2047, [8] := 2047, [9] := 2047, [10] := 2047, [11] := 2047, [12] := 2047, [13] := 2047, [14] := 2047, [15] := 2047, [16] := 2047, [17] := 2047, [18] := 2047, [19] := 2047, [20] := 2047, [21] := 2047, [22] := 2047, [23] := 2047, [24] := 2047, [25] := 2047, [26] := 2047, [27] := 2047, [28] := 2047, [29] := 2047, [30] := 2047, [31] := 2047, [32] := 2047, [33] := 2047, [34] := 2047, [35] := 2047, [36] := 2047, [37] := 2047, [38] := 2047, [39] := 2047, [40] := 2047, [41] := 2047, [42] := 2047, [43] := 2047, [44] := 2047, [45] := 2047, [46] := 2047, [47] := 2047, [48] := 2047, [49] := 2047);
   A_SUM : DINT := 102350;
   A_TOP : SINT := 11;
   AB_N : SINT := 50;
   ACMI_ST1_QAB_VAR : REAL := 11.303459;
   ACMI_ST1_QBA_VAR : REAL := 11.533579;
   ACMI_ST2_QAB_VAR : REAL := 11.294024;
   ACMI_ST2_QBA_VAR : REAL := 11.572626;
   ADC1 : COUNTER;
   B_AVG : REAL := 45.38;
   B_HIST : DINT[50] := ([0] := 45, [1] := 37, [2] := 37, [3] := 52, [4] := 50, [5] := 44, [6] := 43, [7] := 37, [8] := 35, [9] := 45, [10] := 58, [11] := 56, [12] := 51, [13] := 53, [14] := 47, [15] := 49, [16] := 46, [17] := 40, [18] := 57, [19] := 58, [20] := 39, [21] := 52, [22] := 47, [23] := 34, [24] := 28, [25] := 60, [26] := 57, [27] := 52, [28] := 38, [29] := 30, [30] := 45, [31] := 27, [32] := 45, [33] := 43, [34] := 40, [35] := 36, [36] := 42, [37] := 45, [38] := 31, [39] := 42, [40] := 62, [41] := 60, [42] := 49, [43] := 42, [44] := 38, [45] := 50, [46] := 30, [47] := 51, [48] := 63, [49] := 51);
   B_SUM : DINT := 2269;
   B_TOP : SINT := 11;
   Bin_Width : REAL := 0.015; {constant}
   C_AVG : REAL := 33.66; {access Read Only}
   C_HIST : DINT[50] := ([0] := 36, [1] := 22, [2] := 51, [3] := 50, [4] := 46, [5] := 40, [6] := 30, [7] := 20, [8] := 51, [9] := 23, [10] := 41, [11] := 36, [12] := 33, [13] := 34, [14] := 28, [15] := 23, [16] := 33, [17] := 45, [18] := 42, [19] := 37, [20] := 28, [21] := 29, [22] := 20, [23] := 35, [24] := 45, [25] := 43, [26] := 33, [27] := 35, [28] := 18, [29] := 20, [30] := 29, [31] := 32, [32] := 27, [33] := 35, [34] := 23, [35] := 22, [36] := 24, [37] := 26, [38] := 18, [39] := 53, [40] := 36, [41] := 46, [42] := 37, [43] := 31, [44] := 22, [45] := 34, [46] := 37, [47] := 41, [48] := 45, [49] := 38); {access Read Only}
   C_SUM : DINT := 1683; {access Read Only}
   C_TOP : SINT := 9; {access Read Only}
   CAL_INIT : BOOL;
   CAL_Zero : DINT[50]; {constant, access Read Only}
   CD_N : SINT := 50; {access Read Only}
   CLR_AB : BOOL := 1;
   CLR_CD : BOOL := 1;
   D_AVG : REAL := 2047.0; {access Read Only}
   D_HIST : DINT[50] := ([0] := 2047, [1] := 2047, [2] := 2047, [3] := 2047, [4] := 2047, [5] := 2047, [6] := 2047, [7] := 2047, [8] := 2047, [9] := 2047, [10] := 2047, [11] := 2047, [12] := 2047, [13] := 2047, [14] := 2047, [15] := 2047, [16] := 2047, [17] := 2047, [18] := 2047, [19] := 2047, [20] := 2047, [21] := 2047, [22] := 2047, [23] := 2047, [24] := 2047, [25] := 2047, [26] := 2047, [27] := 2047, [28] := 2047, [29] := 2047, [30] := 2047, [31] := 2047, [32] := 2047, [33] := 2047, [34] := 2047, [35] := 2047, [36] := 2047, [37] := 2047, [38] := 2047, [39] := 2047, [40] := 2047, [41] := 2047, [42] := 2047, [43] := 2047, [44] := 2047, [45] := 2047, [46] := 2047, [47] := 2047, [48] := 2047, [49] := 2047); {access Read Only}
   D_SUM : DINT := 102350; {access Read Only}
   D_TOP : SINT := 9; {access Read Only}
   EmptyHist : DINT[31]; {constant}
   H : DINT[31] := ([30] := 200);
   HCntr : REAL := 15.98;
   Index : INT := 30;
   INDX : INT[500] := ([0] := 30, [1] := 30, [2] := 30, [3] := 30, [4] := 30, [5] := 30, [6] := 30, [7] := 30, [8] := 30, [9] := 30, [10] := 30, [11] := 30, [12] := 30, [13] := 30, [14] := 30, [15] := 30, [16] := 30, [17] := 30, [18] := 30, [19] := 30, [20] := 30, [21] := 30, [22] := 30, [23] := 30, [24] := 30, [25] := 30, [26] := 30, [27] := 30, [28] := 30, [29] := 30, [30] := 30, [31] := 30, [32] := 30, [33] := 30, [34] := 30, [35] := 30, [36] := 30, [37] := 30, [38] := 30, [39] := 30, [40] := 30, [41] := 30, [42] := 30, [43] := 30, [44] := 30, [45] := 30, [46] := 30, [47] := 30, [48] := 30, [49] := 30, [50] := 30, [51] := 30, [52] := 30, [53] := 30, [54] := 30, [55] := 30, [56] := 30, [57] := 30, [58] := 30, [59] := 30,
        [60] := 30, [61] := 30, [62] := 30, [63] := 30, [64] := 30, [65] := 30, [66] := 30, [67] := 30, [68] := 30, [69] := 30, [70] := 30, [71] := 30, [72] := 30, [73] := 30, [74] := 30, [75] := 30, [76] := 30, [77] := 30, [78] := 30, [79] := 30, [80] := 30, [81] := 30, [82] := 30, [83] := 30, [84] := 30, [85] := 30, [86] := 30, [87] := 30, [88] := 30, [89] := 30, [90] := 30, [91] := 30, [92] := 30, [93] := 30, [94] := 30, [95] := 30, [96] := 30, [97] := 30, [98] := 30, [99] := 30, [100] := 30, [101] := 30, [102] := 30, [103] := 30, [104] := 30, [105] := 30, [106] := 30, [107] := 30, [108] := 30, [109] := 30, [110] := 30, [111] := 30, [112] := 30, [113] := 30, [114] := 30, [115] := 30, [116] := 30, [117] := 30, [118] := 30, [119] := 30,
        [120] := 30, [121] := 30, [122] := 30, [123] := 30, [124] := 30, [125] := 30, [126] := 30, [127] := 30, [128] := 30, [129] := 30, [130] := 30, [131] := 30, [132] := 30, [133] := 30, [134] := 30, [135] := 30, [136] := 30, [137] := 30, [138] := 30, [139] := 30, [140] := 30, [141] := 30, [142] := 30, [143] := 30, [144] := 30, [145] := 30, [146] := 30, [147] := 30, [148] := 30, [149] := 30, [150] := 30, [151] := 30, [152] := 30, [153] := 30, [154] := 30, [155] := 30, [156] := 30, [157] := 30, [158] := 30, [159] := 30, [160] := 30, [161] := 30, [162] := 30, [163] := 30, [164] := 30, [165] := 30, [166] := 30, [167] := 30, [168] := 30, [169] := 30, [170] := 30, [171] := 30, [172] := 30, [173] := 30, [174] := 30, [175] := 30, [176] := 30, [177] := 30, [178] := 30, [179] := 30,
        [180] := 30, [181] := 30, [182] := 30, [183] := 30, [184] := 30, [185] := 30, [186] := 30, [187] := 30, [188] := 30, [189] := 30, [190] := 30, [191] := 30, [192] := 30, [193] := 30, [194] := 30, [195] := 30, [196] := 30, [197] := 30, [198] := 30, [199] := 30, [200] := -1, [201] := -1, [202] := -1, [203] := -1, [204] := -1, [205] := -1, [206] := -1, [207] := -1, [208] := -1, [209] := -1, [210] := -1, [211] := -1, [212] := -1, [213] := -1, [214] := -1, [215] := -1, [216] := -1, [217] := -1, [218] := -1, [219] := -1, [220] := -1, [221] := -1, [222] := -1, [223] := -1, [224] := -1, [225] := -1, [226] := -1, [227] := -1, [228] := -1, [229] := -1, [230] := -1, [231] := -1, [232] := -1, [233] := -1, [234] := -1, [235] := -1, [236] := -1, [237] := -1, [238] := -1, [239] := -1,
        [240] := -1, [241] := -1, [242] := -1, [243] := -1, [244] := -1, [245] := -1, [246] := -1, [247] := -1, [248] := -1, [249] := -1, [250] := -1, [251] := -1, [252] := -1, [253] := -1, [254] := -1, [255] := -1, [256] := -1, [257] := -1, [258] := -1, [259] := -1, [260] := -1, [261] := -1, [262] := -1, [263] := -1, [264] := -1, [265] := -1, [266] := -1, [267] := -1, [268] := -1, [269] := -1, [270] := -1, [271] := -1, [272] := -1, [273] := -1, [274] := -1, [275] := -1, [276] := -1, [277] := -1, [278] := -1, [279] := -1, [280] := -1, [281] := -1, [282] := -1, [283] := -1, [284] := -1, [285] := -1, [286] := -1, [287] := -1, [288] := -1, [289] := -1, [290] := -1, [291] := -1, [292] := -1, [293] := -1, [294] := -1, [295] := -1, [296] := -1, [297] := -1, [298] := -1, [299] := -1,
        [300] := -1, [301] := -1);
   Init_INDX : INT[500] := ([0] := -1, [1] := -1, [2] := -1, [3] := -1, [4] := -1, [5] := -1, [6] := -1, [7] := -1, [8] := -1, [9] := -1, [10] := -1, [11] := -1, [12] := -1, [13] := -1, [14] := -1, [15] := -1, [16] := -1, [17] := -1, [18] := -1, [19] := -1, [20] := -1, [21] := -1, [22] := -1, [23] := -1, [24] := -1, [25] := -1, [26] := -1, [27] := -1, [28] := -1, [29] := -1, [30] := -1, [31] := -1, [32] := -1, [33] := -1, [34] := -1, [35] := -1, [36] := -1, [37] := -1, [38] := -1, [39] := -1, [40] := -1, [41] := -1, [42] := -1, [43] := -1, [44] := -1, [45] := -1, [46] := -1, [47] := -1, [48] := -1, [49] := -1, [50] := -1, [51] := -1, [52] := -1, [53] := -1, [54] := -1, [55] := -1, [56] := -1, [57] := -1, [58] := -1, [59] := -1,
        [60] := -1, [61] := -1, [62] := -1, [63] := -1, [64] := -1, [65] := -1, [66] := -1, [67] := -1, [68] := -1, [69] := -1, [70] := -1, [71] := -1, [72] := -1, [73] := -1, [74] := -1, [75] := -1, [76] := -1, [77] := -1, [78] := -1, [79] := -1, [80] := -1, [81] := -1, [82] := -1, [83] := -1, [84] := -1, [85] := -1, [86] := -1, [87] := -1, [88] := -1, [89] := -1, [90] := -1, [91] := -1, [92] := -1, [93] := -1, [94] := -1, [95] := -1, [96] := -1, [97] := -1, [98] := -1, [99] := -1, [100] := -1, [101] := -1, [102] := -1, [103] := -1, [104] := -1, [105] := -1, [106] := -1, [107] := -1, [108] := -1, [109] := -1, [110] := -1, [111] := -1, [112] := -1, [113] := -1, [114] := -1, [115] := -1, [116] := -1, [117] := -1, [118] := -1, [119] := -1,
        [120] := -1, [121] := -1, [122] := -1, [123] := -1, [124] := -1, [125] := -1, [126] := -1, [127] := -1, [128] := -1, [129] := -1, [130] := -1, [131] := -1, [132] := -1, [133] := -1, [134] := -1, [135] := -1, [136] := -1, [137] := -1, [138] := -1, [139] := -1, [140] := -1, [141] := -1, [142] := -1, [143] := -1, [144] := -1, [145] := -1, [146] := -1, [147] := -1, [148] := -1, [149] := -1, [150] := -1, [151] := -1, [152] := -1, [153] := -1, [154] := -1, [155] := -1, [156] := -1, [157] := -1, [158] := -1, [159] := -1, [160] := -1, [161] := -1, [162] := -1, [163] := -1, [164] := -1, [165] := -1, [166] := -1, [167] := -1, [168] := -1, [169] := -1, [170] := -1, [171] := -1, [172] := -1, [173] := -1, [174] := -1, [175] := -1, [176] := -1, [177] := -1, [178] := -1, [179] := -1,
        [180] := -1, [181] := -1, [182] := -1, [183] := -1, [184] := -1, [185] := -1, [186] := -1, [187] := -1, [188] := -1, [189] := -1, [190] := -1, [191] := -1, [192] := -1, [193] := -1, [194] := -1, [195] := -1, [196] := -1, [197] := -1, [198] := -1, [199] := -1, [200] := -1, [201] := -1, [202] := -1, [203] := -1, [204] := -1, [205] := -1, [206] := -1, [207] := -1, [208] := -1, [209] := -1, [210] := -1, [211] := -1, [212] := -1, [213] := -1, [214] := -1, [215] := -1, [216] := -1, [217] := -1, [218] := -1, [219] := -1, [220] := -1, [221] := -1, [222] := -1, [223] := -1, [224] := -1, [225] := -1, [226] := -1, [227] := -1, [228] := -1, [229] := -1, [230] := -1, [231] := -1, [232] := -1, [233] := -1, [234] := -1, [235] := -1, [236] := -1, [237] := -1, [238] := -1, [239] := -1,
        [240] := -1, [241] := -1, [242] := -1, [243] := -1, [244] := -1, [245] := -1, [246] := -1, [247] := -1, [248] := -1, [249] := -1, [250] := -1, [251] := -1, [252] := -1, [253] := -1, [254] := -1, [255] := -1, [256] := -1, [257] := -1, [258] := -1, [259] := -1, [260] := -1, [261] := -1, [262] := -1, [263] := -1, [264] := -1, [265] := -1, [266] := -1, [267] := -1, [268] := -1, [269] := -1, [270] := -1, [271] := -1, [272] := -1, [273] := -1, [274] := -1, [275] := -1, [276] := -1, [277] := -1, [278] := -1, [279] := -1, [280] := -1, [281] := -1, [282] := -1, [283] := -1, [284] := -1, [285] := -1, [286] := -1, [287] := -1, [288] := -1, [289] := -1, [290] := -1, [291] := -1, [292] := -1, [293] := -1, [294] := -1, [295] := -1, [296] := -1, [297] := -1, [298] := -1, [299] := -1,
        [300] := -1, [301] := -1); {constant}
   Init_Stats : BOOL := 1;
   ITOP : INT := 44;
   old_index : DINT := 30;
   Proc_ST1AB : BOOL;
   Proc_ST1BA : BOOL := 1;
   Proc_ST2AB : BOOL := 1;
   Proc_ST2BA : BOOL;
   Qavg : REAL := 18.345718;
   Qmax : REAL := 19.713;
   Qmin : REAL := -17.572;
   QnC : REAL := 19.062;
   QpC : DINT := 19062;
   Qstd : REAL := 3360.6584;
   Qvar : REAL := 11.294024;
   Rbit : BOOL := 1;
   REbit : BOOL;
   SSID : STRING := 'D72F2CAC'; {access Read Only}
   SSID_Exists : INT := 1; {access Read Only}
   SSID_Locked : INT := 1; {access Read Only}
   ST1_HCntr : REAL := 0.58;
   ST1_QAB_INDX : INT[500] := ([0] := 30, [1] := 30, [2] := 30, [3] := 30, [4] := 30, [5] := 30, [6] := 30, [7] := 30, [8] := 30, [9] := 30, [10] := 30, [11] := 30, [12] := 30, [13] := 30, [14] := 30, [15] := 30, [16] := 30, [17] := 30, [18] := 30, [19] := 30, [20] := 30, [21] := 30, [22] := 30, [23] := 30, [24] := 30, [25] := 30, [26] := 30, [27] := 30, [28] := 30, [29] := 30, [30] := 30, [31] := 30, [32] := 30, [33] := 30, [34] := 30, [35] := 30, [36] := 30, [37] := 30, [38] := 30, [39] := 30, [40] := 30, [41] := 30, [42] := 30, [43] := 30, [44] := 30, [45] := 30, [46] := 30, [47] := 30, [48] := 30, [49] := 30, [50] := 30, [51] := 30, [52] := 30, [53] := 30, [54] := 30, [55] := 30, [56] := 30, [57] := 30, [58] := 30, [59] := 30,
        [60] := 30, [61] := 30, [62] := 30, [63] := 30, [64] := 30, [65] := 30, [66] := 30, [67] := 30, [68] := 30, [69] := 30, [70] := 30, [71] := 30, [72] := 30, [73] := 30, [74] := 30, [75] := 30, [76] := 30, [77] := 30, [78] := 30, [79] := 30, [80] := 30, [81] := 30, [82] := 30, [83] := 30, [84] := 30, [85] := 30, [86] := 30, [87] := 30, [88] := 30, [89] := 30, [90] := 30, [91] := 30, [92] := 30, [93] := 30, [94] := 30, [95] := 30, [96] := 30, [97] := 30, [98] := 30, [99] := 30, [100] := 30, [101] := 30, [102] := 30, [103] := 30, [104] := 30, [105] := 30, [106] := 30, [107] := 30, [108] := 30, [109] := 30, [110] := 30, [111] := 30, [112] := 30, [113] := 30, [114] := 30, [115] := 30, [116] := 30, [117] := 30, [118] := 30, [119] := 30,
        [120] := 30, [121] := 30, [122] := 30, [123] := 30, [124] := 30, [125] := 30, [126] := 30, [127] := 30, [128] := 30, [129] := 30, [130] := 30, [131] := 30, [132] := 30, [133] := 30, [134] := 30, [135] := 30, [136] := 30, [137] := 30, [138] := 30, [139] := 30, [140] := 30, [141] := 30, [142] := 30, [143] := 30, [144] := 30, [145] := 30, [146] := 30, [147] := 30, [148] := 30, [149] := 30, [150] := 30, [151] := 30, [152] := 30, [153] := 30, [154] := 30, [155] := 30, [156] := 30, [157] := 30, [158] := 30, [159] := 30, [160] := 30, [161] := 30, [162] := 30, [163] := 30, [164] := 30, [165] := 30, [166] := 30, [167] := 30, [168] := 30, [169] := 30, [170] := 30, [171] := 30, [172] := 30, [173] := 30, [174] := 30, [175] := 30, [176] := 30, [177] := 30, [178] := 30, [179] := 30,
        [180] := 30, [181] := 30, [182] := 30, [183] := 30, [184] := 30, [185] := 30, [186] := 30, [187] := 30, [188] := 30, [189] := 30, [190] := 30, [191] := 30, [192] := 30, [193] := 30, [194] := 30, [195] := 30, [196] := 30, [197] := 30, [198] := 30, [199] := 30, [200] := -1, [201] := -1, [202] := -1, [203] := -1, [204] := -1, [205] := -1, [206] := -1, [207] := -1, [208] := -1, [209] := -1, [210] := -1, [211] := -1, [212] := -1, [213] := -1, [214] := -1, [215] := -1, [216] := -1, [217] := -1, [218] := -1, [219] := -1, [220] := -1, [221] := -1, [222] := -1, [223] := -1, [224] := -1, [225] := -1, [226] := -1, [227] := -1, [228] := -1, [229] := -1, [230] := -1, [231] := -1, [232] := -1, [233] := -1, [234] := -1, [235] := -1, [236] := -1, [237] := -1, [238] := -1, [239] := -1,
        [240] := -1, [241] := -1, [242] := -1, [243] := -1, [244] := -1, [245] := -1, [246] := -1, [247] := -1, [248] := -1, [249] := -1, [250] := -1, [251] := -1, [252] := -1, [253] := -1, [254] := -1, [255] := -1, [256] := -1, [257] := -1, [258] := -1, [259] := -1, [260] := -1, [261] := -1, [262] := -1, [263] := -1, [264] := -1, [265] := -1, [266] := -1, [267] := -1, [268] := -1, [269] := -1, [270] := -1, [271] := -1, [272] := -1, [273] := -1, [274] := -1, [275] := -1, [276] := -1, [277] := -1, [278] := -1, [279] := -1, [280] := -1, [281] := -1, [282] := -1, [283] := -1, [284] := -1, [285] := -1, [286] := -1, [287] := -1, [288] := -1, [289] := -1, [290] := -1, [291] := -1, [292] := -1, [293] := -1, [294] := -1, [295] := -1, [296] := -1, [297] := -1, [298] := -1, [299] := -1,
        [300] := -1, [301] := -1);
   ST1_QAB_INDX_TOP : INT := 43;
   ST1_QBA_INDX : INT[500] := ([0] := 30, [1] := 30, [2] := 30, [3] := 30, [4] := 30, [5] := 30, [6] := 30, [7] := 30, [8] := 30, [9] := 30, [10] := 30, [11] := 30, [12] := 30, [13] := 30, [14] := 30, [15] := 30, [16] := 30, [17] := 30, [18] := 30, [19] := 30, [20] := 30, [21] := 30, [22] := 30, [23] := 30, [24] := 30, [25] := 30, [26] := 30, [27] := 30, [28] := 30, [29] := 30, [30] := 30, [31] := 30, [32] := 30, [33] := 30, [34] := 30, [35] := 30, [36] := 30, [37] := 30, [38] := 30, [39] := 30, [40] := 30, [41] := 30, [42] := 30, [43] := 30, [44] := 30, [45] := 30, [46] := 30, [47] := 30, [48] := 30, [49] := 30, [50] := 30, [51] := 30, [52] := 30, [53] := 30, [54] := 30, [55] := 30, [56] := 30, [57] := 30, [58] := 30, [59] := 30,
        [60] := 30, [61] := 30, [62] := 30, [63] := 30, [64] := 30, [65] := 30, [66] := 30, [67] := 30, [68] := 30, [69] := 30, [70] := 30, [71] := 30, [72] := 30, [73] := 30, [74] := 30, [75] := 30, [76] := 30, [77] := 30, [78] := 30, [79] := 30, [80] := 30, [81] := 30, [82] := 30, [83] := 30, [84] := 30, [85] := 30, [86] := 30, [87] := 30, [88] := 30, [89] := 30, [90] := 30, [91] := 30, [92] := 30, [93] := 30, [94] := 30, [95] := 30, [96] := 30, [97] := 30, [98] := 30, [99] := 30, [100] := 30, [101] := 30, [102] := 30, [103] := 30, [104] := 30, [105] := 30, [106] := 30, [107] := 30, [108] := 30, [109] := 30, [110] := 30, [111] := 30, [112] := 30, [113] := 30, [114] := 30, [115] := 30, [116] := 30, [117] := 30, [118] := 30, [119] := 30,
        [120] := 30, [121] := 30, [122] := 30, [123] := 30, [124] := 30, [125] := 30, [126] := 30, [127] := 30, [128] := 30, [129] := 30, [130] := 30, [131] := 30, [132] := 30, [133] := 30, [134] := 30, [135] := 30, [136] := 30, [137] := 30, [138] := 30, [139] := 30, [140] := 30, [141] := 30, [142] := 30, [143] := 30, [144] := 30, [145] := 30, [146] := 30, [147] := 30, [148] := 30, [149] := 30, [150] := 30, [151] := 30, [152] := 30, [153] := 30, [154] := 30, [155] := 30, [156] := 30, [157] := 30, [158] := 30, [159] := 30, [160] := 30, [161] := 30, [162] := 30, [163] := 30, [164] := 30, [165] := 30, [166] := 30, [167] := 30, [168] := 30, [169] := 30, [170] := 30, [171] := 30, [172] := 30, [173] := 30, [174] := 30, [175] := 30, [176] := 30, [177] := 30, [178] := 30, [179] := 30,
        [180] := 30, [181] := 30, [182] := 30, [183] := 30, [184] := 30, [185] := 30, [186] := 30, [187] := 30, [188] := 30, [189] := 30, [190] := 30, [191] := 30, [192] := 30, [193] := 30, [194] := 30, [195] := 30, [196] := 30, [197] := 30, [198] := 30, [199] := 30, [200] := -1, [201] := -1, [202] := -1, [203] := -1, [204] := -1, [205] := -1, [206] := -1, [207] := -1, [208] := -1, [209] := -1, [210] := -1, [211] := -1, [212] := -1, [213] := -1, [214] := -1, [215] := -1, [216] := -1, [217] := -1, [218] := -1, [219] := -1, [220] := -1, [221] := -1, [222] := -1, [223] := -1, [224] := -1, [225] := -1, [226] := -1, [227] := -1, [228] := -1, [229] := -1, [230] := -1, [231] := -1, [232] := -1, [233] := -1, [234] := -1, [235] := -1, [236] := -1, [237] := -1, [238] := -1, [239] := -1,
        [240] := -1, [241] := -1, [242] := -1, [243] := -1, [244] := -1, [245] := -1, [246] := -1, [247] := -1, [248] := -1, [249] := -1, [250] := -1, [251] := -1, [252] := -1, [253] := -1, [254] := -1, [255] := -1, [256] := -1, [257] := -1, [258] := -1, [259] := -1, [260] := -1, [261] := -1, [262] := -1, [263] := -1, [264] := -1, [265] := -1, [266] := -1, [267] := -1, [268] := -1, [269] := -1, [270] := -1, [271] := -1, [272] := -1, [273] := -1, [274] := -1, [275] := -1, [276] := -1, [277] := -1, [278] := -1, [279] := -1, [280] := -1, [281] := -1, [282] := -1, [283] := -1, [284] := -1, [285] := -1, [286] := -1, [287] := -1, [288] := -1, [289] := -1, [290] := -1, [291] := -1, [292] := -1, [293] := -1, [294] := -1, [295] := -1, [296] := -1, [297] := -1, [298] := -1, [299] := -1,
        [300] := -1, [301] := -1);
   ST1_QBA_INDX_TOP : INT := 44;
   ST2_HCntr : REAL := 15.98;
   ST2_QAB_INDX : INT[500] := ([0] := 30, [1] := 30, [2] := 30, [3] := 30, [4] := 30, [5] := 30, [6] := 30, [7] := 30, [8] := 30, [9] := 30, [10] := 30, [11] := 30, [12] := 30, [13] := 30, [14] := 30, [15] := 30, [16] := 30, [17] := 30, [18] := 30, [19] := 30, [20] := 30, [21] := 30, [22] := 30, [23] := 30, [24] := 30, [25] := 30, [26] := 30, [27] := 30, [28] := 30, [29] := 30, [30] := 30, [31] := 30, [32] := 30, [33] := 30, [34] := 30, [35] := 30, [36] := 30, [37] := 30, [38] := 30, [39] := 30, [40] := 30, [41] := 30, [42] := 30, [43] := 30, [44] := 30, [45] := 30, [46] := 30, [47] := 30, [48] := 30, [49] := 30, [50] := 30, [51] := 30, [52] := 30, [53] := 30, [54] := 30, [55] := 30, [56] := 30, [57] := 30, [58] := 30, [59] := 30,
        [60] := 30, [61] := 30, [62] := 30, [63] := 30, [64] := 30, [65] := 30, [66] := 30, [67] := 30, [68] := 30, [69] := 30, [70] := 30, [71] := 30, [72] := 30, [73] := 30, [74] := 30, [75] := 30, [76] := 30, [77] := 30, [78] := 30, [79] := 30, [80] := 30, [81] := 30, [82] := 30, [83] := 30, [84] := 30, [85] := 30, [86] := 30, [87] := 30, [88] := 30, [89] := 30, [90] := 30, [91] := 30, [92] := 30, [93] := 30, [94] := 30, [95] := 30, [96] := 30, [97] := 30, [98] := 30, [99] := 30, [100] := 30, [101] := 30, [102] := 30, [103] := 30, [104] := 30, [105] := 30, [106] := 30, [107] := 30, [108] := 30, [109] := 30, [110] := 30, [111] := 30, [112] := 30, [113] := 30, [114] := 30, [115] := 30, [116] := 30, [117] := 30, [118] := 30, [119] := 30,
        [120] := 30, [121] := 30, [122] := 30, [123] := 30, [124] := 30, [125] := 30, [126] := 30, [127] := 30, [128] := 30, [129] := 30, [130] := 30, [131] := 30, [132] := 30, [133] := 30, [134] := 30, [135] := 30, [136] := 30, [137] := 30, [138] := 30, [139] := 30, [140] := 30, [141] := 30, [142] := 30, [143] := 30, [144] := 30, [145] := 30, [146] := 30, [147] := 30, [148] := 30, [149] := 30, [150] := 30, [151] := 30, [152] := 30, [153] := 30, [154] := 30, [155] := 30, [156] := 30, [157] := 30, [158] := 30, [159] := 30, [160] := 30, [161] := 30, [162] := 30, [163] := 30, [164] := 30, [165] := 30, [166] := 30, [167] := 30, [168] := 30, [169] := 30, [170] := 30, [171] := 30, [172] := 30, [173] := 30, [174] := 30, [175] := 30, [176] := 30, [177] := 30, [178] := 30, [179] := 30,
        [180] := 30, [181] := 30, [182] := 30, [183] := 30, [184] := 30, [185] := 30, [186] := 30, [187] := 30, [188] := 30, [189] := 30, [190] := 30, [191] := 30, [192] := 30, [193] := 30, [194] := 30, [195] := 30, [196] := 30, [197] := 30, [198] := 30, [199] := 30, [200] := -1, [201] := -1, [202] := -1, [203] := -1, [204] := -1, [205] := -1, [206] := -1, [207] := -1, [208] := -1, [209] := -1, [210] := -1, [211] := -1, [212] := -1, [213] := -1, [214] := -1, [215] := -1, [216] := -1, [217] := -1, [218] := -1, [219] := -1, [220] := -1, [221] := -1, [222] := -1, [223] := -1, [224] := -1, [225] := -1, [226] := -1, [227] := -1, [228] := -1, [229] := -1, [230] := -1, [231] := -1, [232] := -1, [233] := -1, [234] := -1, [235] := -1, [236] := -1, [237] := -1, [238] := -1, [239] := -1,
        [240] := -1, [241] := -1, [242] := -1, [243] := -1, [244] := -1, [245] := -1, [246] := -1, [247] := -1, [248] := -1, [249] := -1, [250] := -1, [251] := -1, [252] := -1, [253] := -1, [254] := -1, [255] := -1, [256] := -1, [257] := -1, [258] := -1, [259] := -1, [260] := -1, [261] := -1, [262] := -1, [263] := -1, [264] := -1, [265] := -1, [266] := -1, [267] := -1, [268] := -1, [269] := -1, [270] := -1, [271] := -1, [272] := -1, [273] := -1, [274] := -1, [275] := -1, [276] := -1, [277] := -1, [278] := -1, [279] := -1, [280] := -1, [281] := -1, [282] := -1, [283] := -1, [284] := -1, [285] := -1, [286] := -1, [287] := -1, [288] := -1, [289] := -1, [290] := -1, [291] := -1, [292] := -1, [293] := -1, [294] := -1, [295] := -1, [296] := -1, [297] := -1, [298] := -1, [299] := -1,
        [300] := -1, [301] := -1);
   ST2_QAB_INDX_TOP : INT := 44;
   ST2_QBA_INDX : INT[500] := ([0] := 30, [1] := 30, [2] := 30, [3] := 30, [4] := 30, [5] := 30, [6] := 30, [7] := 30, [8] := 30, [9] := 30, [10] := 30, [11] := 30, [12] := 30, [13] := 30, [14] := 30, [15] := 30, [16] := 30, [17] := 30, [18] := 30, [19] := 30, [20] := 30, [21] := 30, [22] := 30, [23] := 30, [24] := 30, [25] := 30, [26] := 30, [27] := 30, [28] := 30, [29] := 30, [30] := 30, [31] := 30, [32] := 30, [33] := 30, [34] := 30, [35] := 30, [36] := 30, [37] := 30, [38] := 30, [39] := 30, [40] := 30, [41] := 30, [42] := 30, [43] := 30, [44] := 30, [45] := 30, [46] := 30, [47] := 30, [48] := 30, [49] := 30, [50] := 30, [51] := 30, [52] := 30, [53] := 30, [54] := 30, [55] := 30, [56] := 30, [57] := 30, [58] := 30, [59] := 30,
        [60] := 30, [61] := 30, [62] := 30, [63] := 30, [64] := 30, [65] := 30, [66] := 30, [67] := 30, [68] := 30, [69] := 30, [70] := 30, [71] := 30, [72] := 30, [73] := 30, [74] := 30, [75] := 30, [76] := 30, [77] := 30, [78] := 30, [79] := 30, [80] := 30, [81] := 30, [82] := 30, [83] := 30, [84] := 30, [85] := 30, [86] := 30, [87] := 30, [88] := 30, [89] := 30, [90] := 30, [91] := 30, [92] := 30, [93] := 30, [94] := 30, [95] := 30, [96] := 30, [97] := 30, [98] := 30, [99] := 30, [100] := 30, [101] := 30, [102] := 30, [103] := 30, [104] := 30, [105] := 30, [106] := 30, [107] := 30, [108] := 30, [109] := 30, [110] := 30, [111] := 30, [112] := 30, [113] := 30, [114] := 30, [115] := 30, [116] := 30, [117] := 30, [118] := 30, [119] := 30,
        [120] := 30, [121] := 30, [122] := 30, [123] := 30, [124] := 30, [125] := 30, [126] := 30, [127] := 30, [128] := 30, [129] := 30, [130] := 30, [131] := 30, [132] := 30, [133] := 30, [134] := 30, [135] := 30, [136] := 30, [137] := 30, [138] := 30, [139] := 30, [140] := 30, [141] := 30, [142] := 30, [143] := 30, [144] := 30, [145] := 30, [146] := 30, [147] := 30, [148] := 30, [149] := 30, [150] := 30, [151] := 30, [152] := 30, [153] := 30, [154] := 30, [155] := 30, [156] := 30, [157] := 30, [158] := 30, [159] := 30, [160] := 30, [161] := 30, [162] := 30, [163] := 30, [164] := 30, [165] := 30, [166] := 30, [167] := 30, [168] := 30, [169] := 30, [170] := 30, [171] := 30, [172] := 30, [173] := 30, [174] := 30, [175] := 30, [176] := 30, [177] := 30, [178] := 30, [179] := 30,
        [180] := 30, [181] := 30, [182] := 30, [183] := 30, [184] := 30, [185] := 30, [186] := 30, [187] := 30, [188] := 30, [189] := 30, [190] := 30, [191] := 30, [192] := 30, [193] := 30, [194] := 30, [195] := 30, [196] := 30, [197] := 30, [198] := 30, [199] := 30, [200] := -1, [201] := -1, [202] := -1, [203] := -1, [204] := -1, [205] := -1, [206] := -1, [207] := -1, [208] := -1, [209] := -1, [210] := -1, [211] := -1, [212] := -1, [213] := -1, [214] := -1, [215] := -1, [216] := -1, [217] := -1, [218] := -1, [219] := -1, [220] := -1, [221] := -1, [222] := -1, [223] := -1, [224] := -1, [225] := -1, [226] := -1, [227] := -1, [228] := -1, [229] := -1, [230] := -1, [231] := -1, [232] := -1, [233] := -1, [234] := -1, [235] := -1, [236] := -1, [237] := -1, [238] := -1, [239] := -1,
        [240] := -1, [241] := -1, [242] := -1, [243] := -1, [244] := -1, [245] := -1, [246] := -1, [247] := -1, [248] := -1, [249] := -1, [250] := -1, [251] := -1, [252] := -1, [253] := -1, [254] := -1, [255] := -1, [256] := -1, [257] := -1, [258] := -1, [259] := -1, [260] := -1, [261] := -1, [262] := -1, [263] := -1, [264] := -1, [265] := -1, [266] := -1, [267] := -1, [268] := -1, [269] := -1, [270] := -1, [271] := -1, [272] := -1, [273] := -1, [274] := -1, [275] := -1, [276] := -1, [277] := -1, [278] := -1, [279] := -1, [280] := -1, [281] := -1, [282] := -1, [283] := -1, [284] := -1, [285] := -1, [286] := -1, [287] := -1, [288] := -1, [289] := -1, [290] := -1, [291] := -1, [292] := -1, [293] := -1, [294] := -1, [295] := -1, [296] := -1, [297] := -1, [298] := -1, [299] := -1,
        [300] := -1, [301] := -1);
   ST2_QBA_INDX_TOP : INT := 195;
   Stat_Size : INT := 200;
   z1 : DINT := 199;
   z2 : REAL := 205.46672;
   z3 : REAL := 3.3606584;
END_VAR

ROUTINE AB_Stats   (* ladder *)
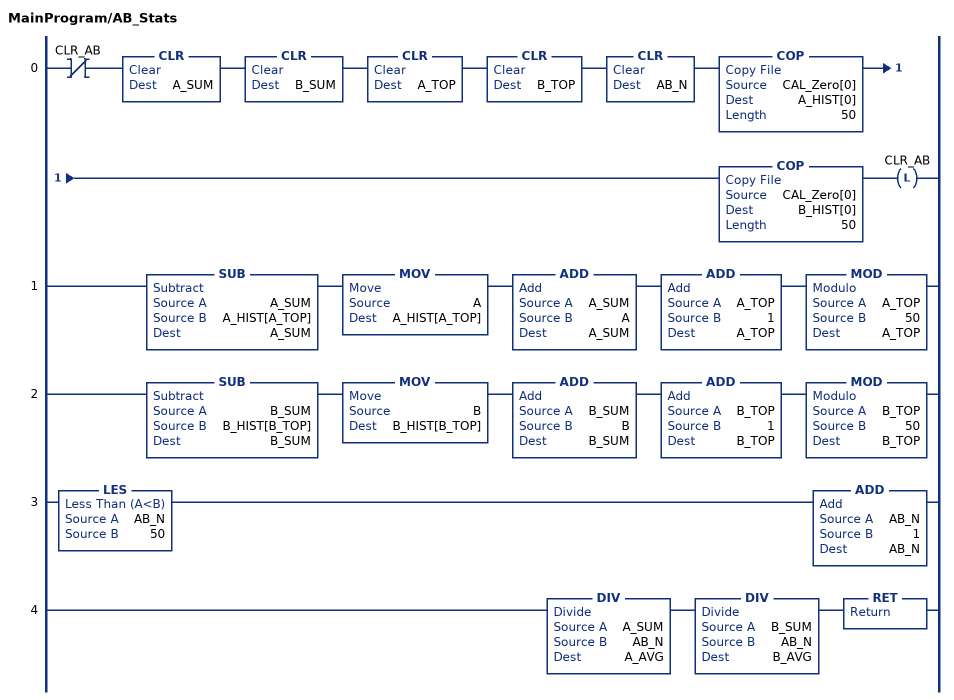
   0: XIO(CLR_AB)CLR(A_SUM)CLR(B_SUM)CLR(A_TOP)CLR(B_TOP)CLR(AB_N)COP(CAL_Zero[0],A_HIST[0],50)COP(CAL_Zero[0],B_HIST[0],50)OTL(CLR_AB);
   1: SUB(A_SUM,A_HIST[A_TOP],A_SUM)MOV(A,A_HIST[A_TOP])ADD(A_SUM,A,A_SUM)ADD(A_TOP,1,A_TOP)MOD(A_TOP,50,A_TOP);
   2: SUB(B_SUM,B_HIST[B_TOP],B_SUM)MOV(B,B_HIST[B_TOP])ADD(B_SUM,B,B_SUM)ADD(B_TOP,1,B_TOP)MOD(B_TOP,50,B_TOP);
   3: LES(AB_N,50)ADD(AB_N,1,AB_N);
   4: DIV(A_SUM,AB_N,A_AVG)DIV(B_SUM,AB_N,B_AVG)RET();
END_ROUTINE

ROUTINE Calc_Histogram   (* ladder *)
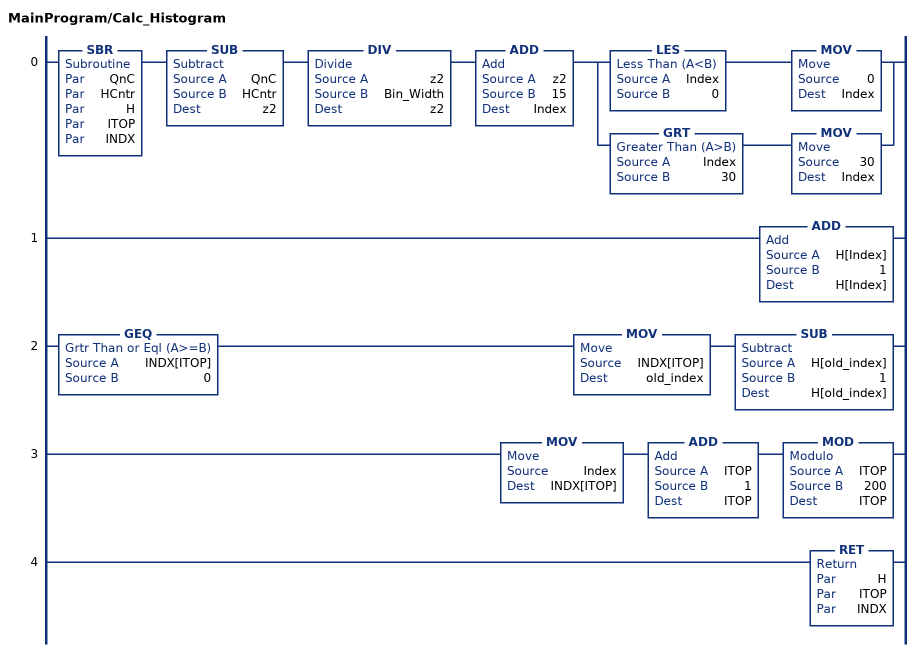
   0: SBR(QnC,HCntr,H,ITOP,INDX)SUB(QnC,HCntr,z2)DIV(z2,Bin_Width,z2)ADD(z2,15,Index)[LES(Index,0) MOV(0,Index) ,GRT(Index,30) MOV(30,Index) ];
   1: ADD(H[Index],1,H[Index]);
   2: GEQ(INDX[ITOP],0)MOV(INDX[ITOP],old_index)SUB(H[old_index],1,H[old_index]);
   3: MOV(Index,INDX[ITOP])ADD(ITOP,1,ITOP)MOD(ITOP,200,ITOP);
   4: RET(H,ITOP,INDX);
END_ROUTINE

ROUTINE Calc_Stats   (* ladder *)
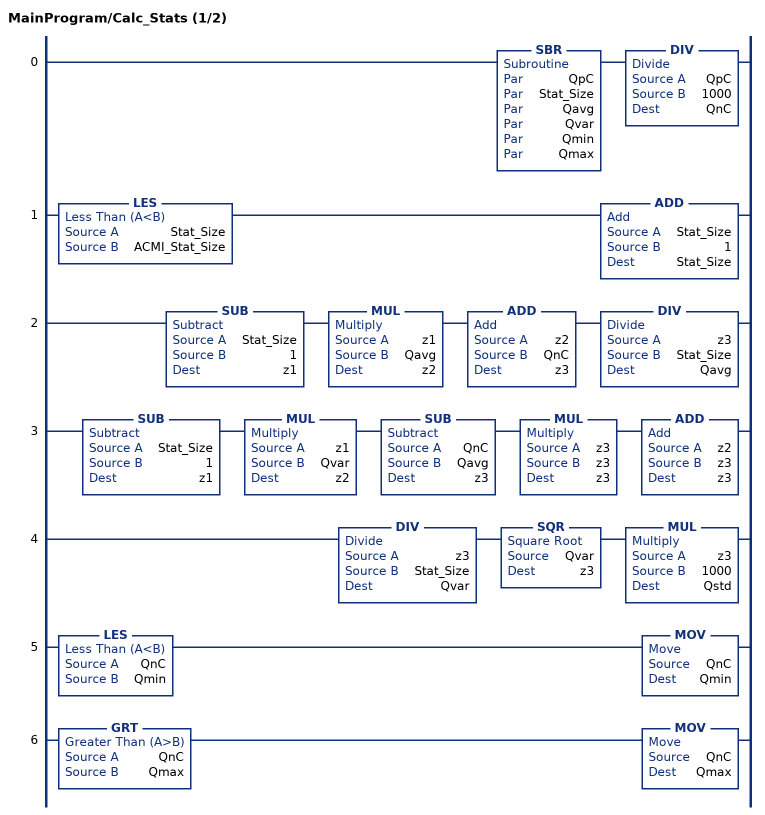
   0: SBR(QpC,Stat_Size,Qavg,Qvar,Qmin,Qmax)DIV(QpC,1000,QnC);
   1: LES(Stat_Size,ACMI_Stat_Size)ADD(Stat_Size,1,Stat_Size);
   2: SUB(Stat_Size,1,z1)MUL(z1,Qavg,z2)ADD(z2,QnC,z3)DIV(z3,Stat_Size,Qavg);
   3: SUB(Stat_Size,1,z1)MUL(z1,Qvar,z2)SUB(QnC,Qavg,z3)MUL(z3,z3,z3)ADD(z2,z3,z3);
   4: DIV(z3,Stat_Size,Qvar)SQR(Qvar,z3)MUL(z3,1000,Qstd);
   5: LES(QnC,Qmin)MOV(QnC,Qmin);
   6: GRT(QnC,Qmax)MOV(QnC,Qmax);
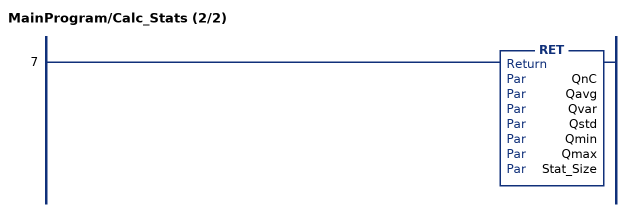
   7: RET(QnC,Qavg,Qvar,Qstd,Qmin,Qmax,Stat_Size);
END_ROUTINE
